LIN {X 0,Y 282.338,Z 551.265,A -85,B 0,C 180,E1 -17007.146,E2 -17007.146} C_VEL
LIN {X 0,Y 282.332,Z 551.855,A -85,B 0,C 180,E1 -17008.574,E2 -17008.574} C_VEL
LIN {X 0,Y 282.332,Z 551.855,A -85,B 0,C 180,E1 -17011.426,E2 -17011.426} C_VEL
LIN {X 0,Y 282.337,Z 551.265,A -85,B 0,C 180,E1 -17012.854,E2 -17012.854} C_VEL
LIN {X 0,Y 282.387,Z 548.814,A -85,B 0,C 180,E1 -17015.713,E2 -17015.713} C_VEL
LIN {X 0,Y 282.678,Z 545.862,A -85,B 0,C 180,E1 -17017.859,E2 -17017.859} C_VEL
LIN {X 0,Y 283.182,Z 541.872,A -85,B 0,C 180,E1 -17020.004,E2 -17020.004} C_VEL
LIN {X 0,Y 283.97,Z 536.74,A -85,B 0,C 180,E1 -17022.144,E2 -17022.144} C_VEL
LIN {X 0,Y 284.964,Z 531.479,A -85,B 0,C 180,E1 -17023.913,E2 -17023.913} C_VEL
LIN {X 0,Y 286.139,Z 525.162,A -85,B 0,C 180,E1 -17025.674,E2 -17025.674} C_VEL
LIN {X 0,Y 287.269,Z 519.212,A -85,B 0,C 180,E1 -17027.072,E2 -17027.072} C_VEL
LIN {X 0,Y 288.401,Z 512.283,A -85,B 0,C 180,E1 -17028.469,E2 -17028.469} C_VEL
LIN {X 0,Y 289.838,Z 504.105,A -85,B 0,C 180,E1 -17029.844,E2 -17029.844} C_VEL
LIN {X 0,Y 291.293,Z 495.598,A -85,B 0,C 180,E1 -17031.031,E2 -17031.031} C_VEL
LIN {X 0,Y 292.626,Z 486.885,A -85,B 0,C 180,E1 -17032.04,E2 -17032.04} C_VEL
LIN {X 0,Y 293.906,Z 477.128,A -85,B 0,C 180,E1 -17032.958,E2 -17032.958} C_VEL
LIN {X 0,Y 294.944,Z 468.339,A -85,B 0,C 180,E1 -17033.616,E2 -17033.616} C_VEL
LIN {X 0,Y 295.883,Z 458.415,A -85,B 0,C 180,E1 -17034.187,E2 -17034.187} C_VEL
LIN {X 0,Y 296.567,Z 448.566,A -85,B 0,C 180,E1 -17034.594,E2 -17034.594} C_VEL
LIN {X 0,Y 297.302,Z 424.442,A -85,B 0,C 180,E1 -17035.216,E2 -17035.216} C_VEL
LIN {X 0,Y 298.17,Z 386.954,A -85,B 0,C 180,E1 -17036.118,E2 -17036.118} C_VEL
LIN {X 0,Y 294.061,Z 364.054,A -85,B 0,C 180,E1 -17037.121,E2 -17037.121} C_VEL
LIN {X 0,Y 290.221,Z 346.945,A -85,B 0,C 180,E1 -17037.974,E2 -17037.974} C_VEL
LIN {X 0,Y 288.061,Z 341.163,A -85,B 0,C 180,E1 -17038.405,E2 -17038.405} C_VEL
LIN {X 0,Y 287.284,Z 336.939,A -85,B 0,C 180,E1 -17040.099,E2 -17040.099} C_VEL
LIN {X 0,Y 285.639,Z 328.615,A -85,B 0,C 180,E1 -17043.785,E2 -17043.785} C_VEL
LIN {X 0,Y 284.339,Z 322.594,A -85,B 0,C 180,E1 -17046.604,E2 -17046.604} C_VEL
LIN {X 0,Y 284.254,Z 322.548,A -85,B 0,C 180,E1 -17050.002,E2 -17050.002} C_VEL
LIN {X 0,Y 284.233,Z 322.579,A -85,B 0,C 180,E1 -17054.187,E2 -17054.187} C_VEL
LIN {X 0,Y 284.27,Z 322.574,A -85,B 0,C 180,E1 -17058.123,E2 -17058.123} C_VEL
LIN {X 0,Y 284.316,Z 322.57,A -85,B 0,C 180,E1 -17062.278,E2 -17062.278} C_VEL
LIN {X 0,Y 284.305,Z 322.55,A -85,B 0,C 180,E1 -17065.349,E2 -17065.349} C_VEL
LIN {X 0,Y 284.29,Z 322.571,A -85,B 0,C 180,E1 -17068.724,E2 -17068.724} C_VEL
LIN {X 0,Y 284.388,Z 322.531,A -85,B 0,C 180,E1 -17072.827,E2 -17072.827} C_VEL
LIN {X 0,Y 284.329,Z 322.564,A -85,B 0,C 180,E1 -17076.703,E2 -17076.703} C_VEL
LIN {X 0,Y 284.393,Z 322.523,A -85,B 0,C 180,E1 -17081.26,E2 -17081.26} C_VEL
LIN {X 0,Y 284.473,Z 322.542,A -85,B 0,C 180,E1 -17084.469,E2 -17084.469} C_VEL
LIN {X 0,Y 284.481,Z 322.525,A -85,B 0,C 180,E1 -17088.6,E2 -17088.6} C_VEL
LIN {X 0,Y 284.632,Z 322.493,A -85,B 0,C 180,E1 -17091.48,E2 -17091.48} C_VEL
LIN {X 0,Y 284.591,Z 322.532,A -85,B 0,C 180,E1 -17094.33,E2 -17094.33} C_VEL
LIN {X 0,Y 284.849,Z 322.475,A -85,B 0,C 180,E1 -17098.585,E2 -17098.585} C_VEL
LIN {X 0,Y 284.848,Z 322.466,A -85,B 0,C 180,E1 -17101.413,E2 -17101.413} C_VEL
LIN {X 0,Y 284.679,Z 322.513,A -85,B 0,C 180,E1 -17107.09,E2 -17107.09} C_VEL
LIN {X 0,Y 284.512,Z 322.504,A -85,B 0,C 180,E1 -17109.956,E2 -17109.956} C_VEL
LIN {X 0,Y 284.471,Z 322.549,A -85,B 0,C 180,E1 -17114.302,E2 -17114.302} C_VEL
LIN {X 0,Y 284.418,Z 322.539,A -85,B 0,C 180,E1 -17117.248,E2 -17117.248} C_VEL
LIN {X 0,Y 284.372,Z 322.535,A -85,B 0,C 180,E1 -17120.242,E2 -17120.242} C_VEL
LIN {X 0,Y 284.362,Z 322.562,A -85,B 0,C 180,E1 -17123.875,E2 -17123.875} C_VEL
LIN {X 0,Y 284.389,Z 322.532,A -85,B 0,C 180,E1 -17127.173,E2 -17127.173} C_VEL
LIN {X 0,Y 284.289,Z 322.574,A -85,B 0,C 180,E1 -17131.274,E2 -17131.274} C_VEL
LIN {X 0,Y 284.355,Z 322.546,A -85,B 0,C 180,E1 -17135.354,E2 -17135.354} C_VEL
LIN {X 0,Y 284.33,Z 322.57,A -85,B 0,C 180,E1 -17138.165,E2 -17138.165} C_VEL
LIN {X 0,Y 284.334,Z 322.56,A -85,B 0,C 180,E1 -17142.14,E2 -17142.14} C_VEL
LIN {X 0,Y 284.29,Z 322.533,A -85,B 0,C 180,E1 -17146.197,E2 -17146.197} C_VEL
LIN {X 0,Y 284.304,Z 322.538,A -85,B 0,C 180,E1 -17150.023,E2 -17150.023} C_VEL
LIN {X 0,Y 284.348,Z 322.545,A -85,B 0,C 180,E1 -17153.617,E2 -17153.617} C_VEL
LIN {X 0,Y 284.302,Z 322.553,A -85,B 0,C 180,E1 -17157.19,E2 -17157.19} C_VEL
LIN {X 0,Y 284.356,Z 322.708,A -85,B 0,C 180,E1 -17160.853,E2 -17160.853} C_VEL
LIN {X 0,Y 284.569,Z 323.646,A -85,B 0,C 180,E1 -17161.126,E2 -17161.126} C_VEL
LIN {X 0,Y 292.585,Z 338.677,A -85,B 0,C 180,E1 -17162.429,E2 -17162.429} C_VEL
LIN {X 0,Y 300.389,Z 349.784,A -85,B 0,C 180,E1 -17163.502,E2 -17163.502} C_VEL
LIN {X 0,Y 308.793,Z 359.275,A -85,B 0,C 180,E1 -17164.601,E2 -17164.601} C_VEL
LIN {X 0,Y 316.905,Z 367.975,A -85,B 0,C 180,E1 -17165.816,E2 -17165.816} C_VEL
LIN {X 0,Y 324.503,Z 375.523,A -85,B 0,C 180,E1 -17167.119,E2 -17167.119} C_VEL
LIN {X 0,Y 332.838,Z 383.472,A -85,B 0,C 180,E1 -17168.723,E2 -17168.723} C_VEL
LIN {X 0,Y 340.839,Z 390.558,A -85,B 0,C 180,E1 -17170.438,E2 -17170.438} C_VEL
LIN {X 0,Y 346.351,Z 394.989,A -85,B 0,C 180,E1 -17171.714,E2 -17171.714} C_VEL
LIN {X 0,Y 353.056,Z 400.728,A -85,B 0,C 180,E1 -17173.434,E2 -17173.434} C_VEL
LIN {X 0,Y 358.555,Z 404.823,A -85,B 0,C 180,E1 -17174.987,E2 -17174.987} C_VEL
LIN {X 0,Y 363.378,Z 408.762,A -85,B 0,C 180,E1 -17176.527,E2 -17176.527} C_VEL
LIN {X 0,Y 368.048,Z 411.828,A -85,B 0,C 180,E1 -17178.185,E2 -17178.185} C_VEL
LIN {X 0,Y 370.508,Z 413.424,A -85,B 0,C 180,E1 -17179.171,E2 -17179.171} C_VEL
LIN {X 0,Y 373.985,Z 416.445,A -85,B 0,C 180,E1 -17180.788,E2 -17180.788} C_VEL
LIN {X 0,Y 377.117,Z 418.611,A -85,B 0,C 180,E1 -17182.504,E2 -17182.504} C_VEL
LIN {X 0,Y 379.745,Z 420.059,A -85,B 0,C 180,E1 -17184.312,E2 -17184.312} C_VEL
LIN {X 0,Y 381.335,Z 420.74,A -85,B 0,C 180,E1 -17185.772,E2 -17185.772} C_VEL
LIN {X 0,Y 382.556,Z 421.148,A -85,B 0,C 180,E1 -17187.355,E2 -17187.355} C_VEL
LIN {X 0,Y 383.208,Z 421.566,A -85,B 0,C 180,E1 -17188.949,E2 -17188.949} C_VEL
LIN {X 0,Y 383.351,Z 421.508,A -85,B 0,C 180,E1 -17190,E2 -17190} C_VEL
LIN {X 0,Y 383.05,Z 421.431,A -85,B 0,C 180,E1 -17191.577,E2 -17191.577} C_VEL
LIN {X 0,Y 382.23,Z 420.939,A -85,B 0,C 180,E1 -17193.162,E2 -17193.162} C_VEL
LIN {X 0,Y 380.5,Z 420.427,A -85,B 0,C 180,E1 -17195.024,E2 -17195.024} C_VEL
LIN {X 0,Y 377.947,Z 419.106,A -85,B 0,C 180,E1 -17196.961,E2 -17196.961} C_VEL
LIN {X 0,Y 374.623,Z 416.948,A -85,B 0,C 180,E1 -17198.885,E2 -17198.885} C_VEL
LIN {X 0,Y 371.032,Z 413.897,A -85,B 0,C 180,E1 -17200.604,E2 -17200.604} C_VEL
LIN {X 0,Y 368.439,Z 411.979,A -85,B 0,C 180,E1 -17201.675,E2 -17201.675} C_VEL
LIN {X 0,Y 364.032,Z 409.248,A -85,B 0,C 180,E1 -17203.256,E2 -17203.256} C_VEL
LIN {X 0,Y 358.884,Z 405.11,A -85,B 0,C 180,E1 -17204.909,E2 -17204.909} C_VEL
LIN {X 0,Y 352.075,Z 399.957,A -85,B 0,C 180,E1 -17206.83,E2 -17206.83} C_VEL
LIN {X 0,Y 345.31,Z 394.26,A -85,B 0,C 180,E1 -17208.53,E2 -17208.53} C_VEL
LIN {X 0,Y 339.058,Z 388.935,A -85,B 0,C 180,E1 -17209.965,E2 -17209.965} C_VEL
LIN {X 0,Y 331.391,Z 382.051,A -85,B 0,C 180,E1 -17211.572,E2 -17211.572} C_VEL
LIN {X 0,Y 323.339,Z 374.346,A -85,B 0,C 180,E1 -17213.096,E2 -17213.096} C_VEL
LIN {X 0,Y 316.273,Z 367.284,A -85,B 0,C 180,E1 -17214.282,E2 -17214.282} C_VEL
LIN {X 0,Y 308.443,Z 358.947,A -85,B 0,C 180,E1 -17215.444,E2 -17215.444} C_VEL
LIN {X 0,Y 299.859,Z 349.077,A -85,B 0,C 180,E1 -17216.568,E2 -17216.568} C_VEL
LIN {X 0,Y 292.259,Z 338.141,A -85,B 0,C 180,E1 -17217.619,E2 -17217.619} C_VEL
LIN {X 0,Y 284.572,Z 323.628,A -85,B 0,C 180,E1 -17218.876,E2 -17218.876} C_VEL
LIN {X 0,Y 284.347,Z 322.628,A -85,B 0,C 180,E1 -17219.19,E2 -17219.19} C_VEL
LIN {X 0,Y 284.3,Z 322.55,A -85,B 0,C 180,E1 -17222.945,E2 -17222.945} C_VEL
LIN {X 0,Y 284.348,Z 322.545,A -85,B 0,C 180,E1 -17226.383,E2 -17226.383} C_VEL
LIN {X 0,Y 284.303,Z 322.537,A -85,B 0,C 180,E1 -17229.994,E2 -17229.994} C_VEL
LIN {X 0,Y 284.287,Z 322.541,A -85,B 0,C 180,E1 -17234.2,E2 -17234.2} C_VEL
LIN {X 0,Y 284.332,Z 322.558,A -85,B 0,C 180,E1 -17238.136,E2 -17238.136} C_VEL
LIN {X 0,Y 284.339,Z 322.567,A -85,B 0,C 180,E1 -17242.272,E2 -17242.272} C_VEL
LIN {X 0,Y 284.317,Z 322.548,A -85,B 0,C 180,E1 -17245.353,E2 -17245.353} C_VEL
LIN {X 0,Y 284.289,Z 322.574,A -85,B 0,C 180,E1 -17248.726,E2 -17248.726} C_VEL
LIN {X 0,Y 284.389,Z 322.532,A -85,B 0,C 180,E1 -17252.827,E2 -17252.827} C_VEL
LIN {X 0,Y 284.359,Z 322.565,A -85,B 0,C 180,E1 -17256.707,E2 -17256.707} C_VEL
LIN {X 0,Y 284.395,Z 322.526,A -85,B 0,C 180,E1 -17261.262,E2 -17261.262} C_VEL
LIN {X 0,Y 284.471,Z 322.547,A -85,B 0,C 180,E1 -17264.47,E2 -17264.47} C_VEL
LIN {X 0,Y 284.48,Z 322.518,A -85,B 0,C 180,E1 -17268.602,E2 -17268.602} C_VEL
LIN {X 0,Y 284.632,Z 322.5,A -85,B 0,C 180,E1 -17271.481,E2 -17271.481} C_VEL
LIN {X 0,Y 284.59,Z 322.533,A -85,B 0,C 180,E1 -17274.332,E2 -17274.332} C_VEL
LIN {X 0,Y 284.848,Z 322.467,A -85,B 0,C 180,E1 -17278.587,E2 -17278.587} C_VEL
LIN {X 0,Y 284.849,Z 322.475,A -85,B 0,C 180,E1 -17281.415,E2 -17281.415} C_VEL
LIN {X 0,Y 284.68,Z 322.508,A -85,B 0,C 180,E1 -17287.091,E2 -17287.091} C_VEL
LIN {X 0,Y 284.513,Z 322.504,A -85,B 0,C 180,E1 -17289.958,E2 -17289.958} C_VEL
LIN {X 0,Y 284.473,Z 322.548,A -85,B 0,C 180,E1 -17294.304,E2 -17294.304} C_VEL
LIN {X 0,Y 284.417,Z 322.529,A -85,B 0,C 180,E1 -17297.25,E2 -17297.25} C_VEL
LIN {X 0,Y 284.379,Z 322.536,A -85,B 0,C 180,E1 -17300.013,E2 -17300.013} C_VEL
LIN {X 0,Y 283.743,Z 322.631,A -85,B 0,C 180,E1 -17301.196,E2 -17301.196} C_VEL
LIN {X 0,Y 280.862,Z 322.997,A -85,B 0,C 180,E1 -17303.121,E2 -17303.121} C_VEL
LIN {X 0,Y 278.406,Z 323.292,A -85,B 0,C 180,E1 -17304.685,E2 -17304.685} C_VEL
LIN {X 0,Y 277.371,Z 323.408,A -85,B 0,C 180,E1 -17305.898,E2 -17305.898} C_VEL
LIN {X 0,Y 277.298,Z 323.414,A -85,B 0,C 180,E1 -17306.309,E2 -17306.309} C_VEL
LIN {X 0,Y 277.269,Z 323.449,A -85,B 0,C 180,E1 -17310.483,E2 -17310.483} C_VEL
LIN {X 0,Y 277.244,Z 323.427,A -85,B 0,C 180,E1 -17313.897,E2 -17313.897} C_VEL
LIN {X 0,Y 277.262,Z 323.448,A -85,B 0,C 180,E1 -17317.471,E2 -17317.471} C_VEL
LIN {X 0,Y 277.208,Z 323.449,A -85,B 0,C 180,E1 -17321.238,E2 -17321.238} C_VEL
LIN {X 0,Y 277.194,Z 323.451,A -85,B 0,C 180,E1 -17325.229,E2 -17325.229} C_VEL
LIN {X 0,Y 277.176,Z 323.43,A -85,B 0,C 180,E1 -17328.759,E2 -17328.759} C_VEL
LIN {X 0,Y 277.301,Z 323.586,A -85,B 0,C 180,E1 -17332.902,E2 -17332.902} C_VEL
LIN {X 0,Y 278.886,Z 330.791,A -85,B 0,C 180,E1 -17336.331,E2 -17336.331} C_VEL
LIN {X 0,Y 280.435,Z 338.656,A -85,B 0,C 180,E1 -17339.92,E2 -17339.92} C_VEL
LIN {X 0,Y 280.841,Z 340.955,A -85,B 0,C 180,E1 -17340.795,E2 -17340.795} C_VEL
LIN {X 0,Y 284.504,Z 350.337,A -85,B 0,C 180,E1 -17341.513,E2 -17341.513} C_VEL
LIN {X 0,Y 289.328,Z 373.325,A -85,B 0,C 180,E1 -17342.656,E2 -17342.656} C_VEL
LIN {X 0,Y 291.893,Z 388.914,A -85,B 0,C 180,E1 -17343.334,E2 -17343.334} C_VEL
LIN {X 0,Y 290.229,Z 447.041,A -85,B 0,C 180,E1 -17344.784,E2 -17344.784} C_VEL
LIN {X 0,Y 289.511,Z 457.348,A -85,B 0,C 180,E1 -17345.197,E2 -17345.197} C_VEL
LIN {X 0,Y 288.58,Z 466.857,A -85,B 0,C 180,E1 -17345.735,E2 -17345.735} C_VEL
LIN {X 0,Y 287.504,Z 475.928,A -85,B 0,C 180,E1 -17346.405,E2 -17346.405} C_VEL
LIN {X 0,Y 286.312,Z 485.06,A -85,B 0,C 180,E1 -17347.257,E2 -17347.257} C_VEL
LIN {X 0,Y 284.893,Z 494.052,A -85,B 0,C 180,E1 -17348.283,E2 -17348.283} C_VEL
LIN {X 0,Y 283.36,Z 502.776,A -85,B 0,C 180,E1 -17349.493,E2 -17349.493} C_VEL
LIN {X 0,Y 281.983,Z 510.168,A -85,B 0,C 180,E1 -17350.717,E2 -17350.717} C_VEL
LIN {X 0,Y 280.589,Z 518.247,A -85,B 0,C 180,E1 -17352.331,E2 -17352.331} C_VEL
LIN {X 0,Y 279.246,Z 524.966,A -85,B 0,C 180,E1 -17353.928,E2 -17353.928} C_VEL
LIN {X 0,Y 278.035,Z 531.284,A -85,B 0,C 180,E1 -17355.733,E2 -17355.733} C_VEL
LIN {X 0,Y 276.992,Z 536.544,A -85,B 0,C 180,E1 -17357.546,E2 -17357.546} C_VEL
LIN {X 0,Y 276.172,Z 541.677,A -85,B 0,C 180,E1 -17359.739,E2 -17359.739} C_VEL
LIN {X 0,Y 275.608,Z 545.667,A -85,B 0,C 180,E1 -17361.938,E2 -17361.938} C_VEL
LIN {X 0,Y 275.254,Z 549.304,A -85,B 0,C 180,E1 -17364.741,E2 -17364.741} C_VEL
LIN {X 0,Y 275.247,Z 551.071,A -85,B 0,C 180,E1 -17367.073,E2 -17367.073} C_VEL
LIN {X 0,Y 275.256,Z 551.662,A -85,B 0,C 180,E1 -17368.537,E2 -17368.537} C_VEL
LIN {X 0,Y 275.256,Z 551.662,A -85,B 0,C 180,E1 -17371.463,E2 -17371.463} C_VEL
LIN {X 0,Y 275.246,Z 551.071,A -85,B 0,C 180,E1 -17372.927,E2 -17372.927} C_VEL
LIN {X 0,Y 275.3,Z 548.619,A -85,B 0,C 180,E1 -17375.861,E2 -17375.861} C_VEL
LIN {X 0,Y 275.607,Z 545.667,A -85,B 0,C 180,E1 -17378.062,E2 -17378.062} C_VEL
LIN {X 0,Y 276.172,Z 541.677,A -85,B 0,C 180,E1 -17380.261,E2 -17380.261} C_VEL
LIN {X 0,Y 276.992,Z 536.544,A -85,B 0,C 180,E1 -17382.454,E2 -17382.454} C_VEL
LIN {X 0,Y 278.03,Z 531.284,A -85,B 0,C 180,E1 -17384.268,E2 -17384.268} C_VEL
LIN {X 0,Y 279.263,Z 524.967,A -85,B 0,C 180,E1 -17386.071,E2 -17386.071} C_VEL
LIN {X 0,Y 280.665,Z 518.016,A -85,B 0,C 180,E1 -17387.718,E2 -17387.718} C_VEL
LIN {X 0,Y 281.664,Z 512.088,A -85,B 0,C 180,E1 -17388.927,E2 -17388.927} C_VEL
LIN {X 0,Y 283.167,Z 503.911,A -85,B 0,C 180,E1 -17390.332,E2 -17390.332} C_VEL
LIN {X 0,Y 284.677,Z 495.404,A -85,B 0,C 180,E1 -17391.544,E2 -17391.544} C_VEL
LIN {X 0,Y 286.062,Z 486.691,A -85,B 0,C 180,E1 -17392.573,E2 -17392.573} C_VEL
LIN {X 0,Y 287.374,Z 476.934,A -85,B 0,C 180,E1 -17393.511,E2 -17393.511} C_VEL
LIN {X 0,Y 288.451,Z 468.145,A -85,B 0,C 180,E1 -17394.181,E2 -17394.181} C_VEL
LIN {X 0,Y 289.426,Z 458.221,A -85,B 0,C 180,E1 -17394.763,E2 -17394.763} C_VEL
LIN {X 0,Y 290.134,Z 448.372,A -85,B 0,C 180,E1 -17395.177,E2 -17395.177} C_VEL
LIN {X 0,Y 290.91,Z 424.264,A -85,B 0,C 180,E1 -17395.81,E2 -17395.81} C_VEL
LIN {X 0,Y 291.819,Z 388.268,A -85,B 0,C 180,E1 -17396.69,E2 -17396.69} C_VEL
LIN {X 0,Y 288.062,Z 366.799,A -85,B 0,C 180,E1 -17397.653,E2 -17397.653} C_VEL
LIN {X 0,Y 284.215,Z 349.549,A -85,B 0,C 180,E1 -17398.54,E2 -17398.54} C_VEL
LIN {X 0,Y 280.84,Z 340.923,A -85,B 0,C 180,E1 -17399.208,E2 -17399.208} C_VEL
LIN {X 0,Y 279.86,Z 335.827,A -85,B 0,C 180,E1 -17401.368,E2 -17401.368} C_VEL
LIN {X 0,Y 278.214,Z 327.795,A -85,B 0,C 180,E1 -17405.077,E2 -17405.077} C_VEL
LIN {X 0,Y 277.285,Z 323.452,A -85,B 0,C 180,E1 -17407.256,E2 -17407.256} C_VEL
LIN {X 0,Y 277.176,Z 323.43,A -85,B 0,C 180,E1 -17411.241,E2 -17411.241} C_VEL
LIN {X 0,Y 277.197,Z 323.447,A -85,B 0,C 180,E1 -17415.226,E2 -17415.226} C_VEL
LIN {X 0,Y 277.22,Z 323.44,A -85,B 0,C 180,E1 -17419.511,E2 -17419.511} C_VEL
LIN {X 0,Y 277.262,Z 323.448,A -85,B 0,C 180,E1 -17422.529,E2 -17422.529} C_VEL
LIN {X 0,Y 277.244,Z 323.427,A -85,B 0,C 180,E1 -17426.103,E2 -17426.103} C_VEL
LIN {X 0,Y 277.259,Z 323.451,A -85,B 0,C 180,E1 -17429.537,E2 -17429.537} C_VEL
LIN {X 0,Y 277.35,Z 323.407,A -85,B 0,C 180,E1 -17432.862,E2 -17432.862} C_VEL
LIN {X 0,Y 277.292,Z 323.44,A -85,B 0,C 180,E1 -17436.075,E2 -17436.075} C_VEL
LIN {X 0,Y 277.337,Z 323.404,A -85,B 0,C 180,E1 -17440.765,E2 -17440.765} C_VEL
LIN {X 0,Y 277.423,Z 323.424,A -85,B 0,C 180,E1 -17445.324,E2 -17445.324} C_VEL
LIN {X 0,Y 277.455,Z 323.383,A -85,B 0,C 180,E1 -17449.786,E2 -17449.786} C_VEL
LIN {X 0,Y 277.634,Z 323.384,A -85,B 0,C 180,E1 -17452.728,E2 -17452.728} C_VEL
LIN {X 0,Y 277.815,Z 323.351,A -85,B 0,C 180,E1 -17458.55,E2 -17458.55} C_VEL
LIN {X 0,Y 277.814,Z 323.342,A -85,B 0,C 180,E1 -17461.449,E2 -17461.449} C_VEL
LIN {X 0,Y 277.634,Z 323.389,A -85,B 0,C 180,E1 -17467.271,E2 -17467.271} C_VEL
LIN {X 0,Y 277.454,Z 323.382,A -85,B 0,C 180,E1 -17470.212,E2 -17470.212} C_VEL
LIN {X 0,Y 277.421,Z 323.429,A -85,B 0,C 180,E1 -17474.674,E2 -17474.674} C_VEL
LIN {X 0,Y 277.337,Z 323.404,A -85,B 0,C 180,E1 -17479.233,E2 -17479.233} C_VEL
LIN {X 0,Y 277.312,Z 323.441,A -85,B 0,C 180,E1 -17484.17,E2 -17484.17} C_VEL
LIN {X 0,Y 277.318,Z 323.412,A -85,B 0,C 180,E1 -17487.504,E2 -17487.504} C_VEL
LIN {X 0,Y 277.265,Z 323.446,A -85,B 0,C 180,E1 -17490.481,E2 -17490.481} C_VEL
LIN {X 0,Y 277.247,Z 323.43,A -85,B 0,C 180,E1 -17493.895,E2 -17493.895} C_VEL
LIN {X 0,Y 277.284,Z 323.447,A -85,B 0,C 180,E1 -17497.466,E2 -17497.466} C_VEL
LIN {X 0,Y 277.257,Z 323.432,A -85,B 0,C 180,E1 -17501.227,E2 -17501.227} C_VEL
LIN {X 0,Y 277.236,Z 323.431,A -85,B 0,C 180,E1 -17505.218,E2 -17505.218} C_VEL
LIN {X 0,Y 277.221,Z 323.408,A -85,B 0,C 180,E1 -17509.511,E2 -17509.511} C_VEL
LIN {X 0,Y 277.281,Z 323.445,A -85,B 0,C 180,E1 -17512.534,E2 -17512.534} C_VEL
LIN {X 0,Y 277.249,Z 323.415,A -85,B 0,C 180,E1 -17516.105,E2 -17516.105} C_VEL
LIN {X 0,Y 277.305,Z 323.576,A -85,B 0,C 180,E1 -17520.073,E2 -17520.073} C_VEL
LIN {X 0,Y 277.556,Z 324.569,A -85,B 0,C 180,E1 -17520.348,E2 -17520.348} C_VEL
LIN {X 0,Y 287.343,Z 342.912,A -85,B 0,C 180,E1 -17521.996,E2 -17521.996} C_VEL
LIN {X 0,Y 294.758,Z 353.585,A -85,B 0,C 180,E1 -17523.052,E2 -17523.052} C_VEL
LIN {X 0,Y 304.118,Z 364.334,A -85,B 0,C 180,E1 -17524.244,E2 -17524.244} C_VEL
LIN {X 0,Y 311.901,Z 372.421,A -85,B 0,C 180,E1 -17525.315,E2 -17525.315} C_VEL
LIN {X 0,Y 318.089,Z 378.443,A -85,B 0,C 180,E1 -17526.266,E2 -17526.266} C_VEL
LIN {X 0,Y 324.451,Z 384.567,A -85,B 0,C 180,E1 -17527.372,E2 -17527.372} C_VEL
LIN {X 0,Y 332.426,Z 391.897,A -85,B 0,C 180,E1 -17528.906,E2 -17528.906} C_VEL
LIN {X 0,Y 340.748,Z 399.068,A -85,B 0,C 180,E1 -17530.692,E2 -17530.692} C_VEL
LIN {X 0,Y 346.278,Z 403.439,A -85,B 0,C 180,E1 -17531.979,E2 -17531.979} C_VEL
LIN {X 0,Y 352.189,Z 408.23,A -85,B 0,C 180,E1 -17533.492,E2 -17533.492} C_VEL
LIN {X 0,Y 356.757,Z 411.554,A -85,B 0,C 180,E1 -17534.763,E2 -17534.763} C_VEL
LIN {X 0,Y 361.884,Z 415.618,A -85,B 0,C 180,E1 -17536.362,E2 -17536.362} C_VEL
LIN {X 0,Y 366.483,Z 418.608,A -85,B 0,C 180,E1 -17537.961,E2 -17537.961} C_VEL
LIN {X 0,Y 369.009,Z 420.209,A -85,B 0,C 180,E1 -17538.942,E2 -17538.942} C_VEL
LIN {X 0,Y 372.659,Z 423.307,A -85,B 0,C 180,E1 -17540.597,E2 -17540.597} C_VEL
LIN {X 0,Y 375.863,Z 425.477,A -85,B 0,C 180,E1 -17542.306,E2 -17542.306} C_VEL
LIN {X 0,Y 378.844,Z 427.104,A -85,B 0,C 180,E1 -17544.299,E2 -17544.299} C_VEL
LIN {X 0,Y 380.515,Z 427.791,A -85,B 0,C 180,E1 -17545.829,E2 -17545.829} C_VEL
LIN {X 0,Y 381.686,Z 428.196,A -85,B 0,C 180,E1 -17547.349,E2 -17547.349} C_VEL
LIN {X 0,Y 382.346,Z 428.597,A -85,B 0,C 180,E1 -17548.947,E2 -17548.947} C_VEL
LIN {X 0,Y 382.488,Z 428.54,A -85,B 0,C 180,E1 -17550,E2 -17550} C_VEL
LIN {X 0,Y 382.181,Z 428.48,A -85,B 0,C 180,E1 -17551.581,E2 -17551.581} C_VEL
LIN {X 0,Y 381.093,Z 427.919,A -85,B 0,C 180,E1 -17553.514,E2 -17553.514} C_VEL
LIN {X 0,Y 379.012,Z 427.165,A -85,B 0,C 180,E1 -17555.563,E2 -17555.563} C_VEL
LIN {X 0,Y 376.179,Z 425.679,A -85,B 0,C 180,E1 -17557.514,E2 -17557.514} C_VEL
LIN {X 0,Y 372.829,Z 423.468,A -85,B 0,C 180,E1 -17559.32,E2 -17559.32} C_VEL
LIN {X 0,Y 369.009,Z 420.204,A -85,B 0,C 180,E1 -17561.058,E2 -17561.058} C_VEL
LIN {X 0,Y 363.501,Z 416.773,A -85,B 0,C 180,E1 -17563.102,E2 -17563.102} C_VEL
LIN {X 0,Y 357.89,Z 412.57,A -85,B 0,C 180,E1 -17564.891,E2 -17564.891} C_VEL
LIN {X 0,Y 353.91,Z 409.438,A -85,B 0,C 180,E1 -17566.037,E2 -17566.037} C_VEL
LIN {X 0,Y 348.023,Z 404.978,A -85,B 0,C 180,E1 -17567.589,E2 -17567.589} C_VEL
LIN {X 0,Y 342.613,Z 400.499,A -85,B 0,C 180,E1 -17568.892,E2 -17568.892} C_VEL
LIN {X 0,Y 336.047,Z 394.971,A -85,B 0,C 180,E1 -17570.342,E2 -17570.342} C_VEL
LIN {X 0,Y 328.448,Z 388.318,A -85,B 0,C 180,E1 -17571.882,E2 -17571.882} C_VEL
LIN {X 0,Y 319.943,Z 380.342,A -85,B 0,C 180,E1 -17573.421,E2 -17573.421} C_VEL
LIN {X 0,Y 312.089,Z 372.639,A -85,B 0,C 180,E1 -17574.656,E2 -17574.656} C_VEL
LIN {X 0,Y 303.673,Z 363.897,A -85,B 0,C 180,E1 -17575.811,E2 -17575.811} C_VEL
LIN {X 0,Y 294.558,Z 353.322,A -85,B 0,C 180,E1 -17576.975,E2 -17576.975} C_VEL
LIN {X 0,Y 287.007,Z 342.377,A -85,B 0,C 180,E1 -17578.055,E2 -17578.055} C_VEL
LIN {X 0,Y 277.549,Z 324.574,A -85,B 0,C 180,E1 -17579.65,E2 -17579.65} C_VEL
LIN {X 0,Y 277.3,Z 323.521,A -85,B 0,C 180,E1 -17579.964,E2 -17579.964} C_VEL
LIN {X 0,Y 277.249,Z 323.415,A -85,B 0,C 180,E1 -17583.895,E2 -17583.895} C_VEL
LIN {X 0,Y 277.281,Z 323.445,A -85,B 0,C 180,E1 -17587.466,E2 -17587.466} C_VEL
LIN {X 0,Y 277.211,Z 323.4,A -85,B 0,C 180,E1 -17591.235,E2 -17591.235} C_VEL
LIN {X 0,Y 277.24,Z 323.44,A -85,B 0,C 180,E1 -17595.217,E2 -17595.217} C_VEL
LIN {X 0,Y 277.288,Z 323.427,A -85,B 0,C 180,E1 -17599.495,E2 -17599.495} C_VEL
LIN {X 0,Y 277.284,Z 323.447,A -85,B 0,C 180,E1 -17602.534,E2 -17602.534} C_VEL
LIN {X 0,Y 277.247,Z 323.43,A -85,B 0,C 180,E1 -17606.105,E2 -17606.105} C_VEL
LIN {X 0,Y 277.255,Z 323.448,A -85,B 0,C 180,E1 -17609.539,E2 -17609.539} C_VEL
LIN {X 0,Y 277.351,Z 323.408,A -85,B 0,C 180,E1 -17612.864,E2 -17612.864} C_VEL
LIN {X 0,Y 277.322,Z 323.439,A -85,B 0,C 180,E1 -17616.08,E2 -17616.08} C_VEL
LIN {X 0,Y 277.337,Z 323.404,A -85,B 0,C 180,E1 -17620.767,E2 -17620.767} C_VEL
LIN {X 0,Y 277.421,Z 323.429,A -85,B 0,C 180,E1 -17625.326,E2 -17625.326} C_VEL
LIN {X 0,Y 277.454,Z 323.382,A -85,B 0,C 180,E1 -17629.788,E2 -17629.788} C_VEL
LIN {X 0,Y 277.634,Z 323.389,A -85,B 0,C 180,E1 -17632.729,E2 -17632.729} C_VEL
LIN {X 0,Y 277.814,Z 323.342,A -85,B 0,C 180,E1 -17638.551,E2 -17638.551} C_VEL
LIN {X 0,Y 277.815,Z 323.351,A -85,B 0,C 180,E1 -17641.45,E2 -17641.45} C_VEL
LIN {X 0,Y 277.634,Z 323.384,A -85,B 0,C 180,E1 -17647.272,E2 -17647.272} C_VEL
LIN {X 0,Y 277.455,Z 323.383,A -85,B 0,C 180,E1 -17650.214,E2 -17650.214} C_VEL
LIN {X 0,Y 277.423,Z 323.424,A -85,B 0,C 180,E1 -17654.676,E2 -17654.676} C_VEL
LIN {X 0,Y 277.337,Z 323.404,A -85,B 0,C 180,E1 -17659.235,E2 -17659.235} C_VEL
LIN {X 0,Y 277.287,Z 323.437,A -85,B 0,C 180,E1 -17664.158,E2 -17664.158} C_VEL
LIN {X 0,Y 277.298,Z 323.414,A -85,B 0,C 180,E1 -17666.309,E2 -17666.309} C_VEL
LIN {X 0,Y 276.64,Z 323.5,A -85,B 0,C 180,E1 -17667.521,E2 -17667.521} C_VEL
LIN {X 0,Y 273.725,Z 323.885,A -85,B 0,C 180,E1 -17669.493,E2 -17669.493} C_VEL
LIN {X 0,Y 271.261,Z 324.194,A -85,B 0,C 180,E1 -17671.096,E2 -17671.096} C_VEL
LIN {X 0,Y 270.239,Z 324.311,A -85,B 0,C 180,E1 -17672.34,E2 -17672.34} C_VEL
LIN {X 0,Y 270.176,Z 324.312,A -85,B 0,C 180,E1 -17672.762,E2 -17672.762} C_VEL
LIN {X 0,Y 270.213,Z 324.327,A -85,B 0,C 180,E1 -17676.743,E2 -17676.743} C_VEL
LIN {X 0,Y 270.167,Z 324.322,A -85,B 0,C 180,E1 -17681.029,E2 -17681.029} C_VEL
LIN {X 0,Y 270.149,Z 324.324,A -85,B 0,C 180,E1 -17684.622,E2 -17684.622} C_VEL
LIN {X 0,Y 270.15,Z 324.322,A -85,B 0,C 180,E1 -17687.439,E2 -17687.439} C_VEL
LIN {X 0,Y 270.232,Z 324.445,A -85,B 0,C 180,E1 -17692.268,E2 -17692.268} C_VEL
LIN {X 0,Y 271.818,Z 331.673,A -85,B 0,C 180,E1 -17695.831,E2 -17695.831} C_VEL
LIN {X 0,Y 273.551,Z 340.382,A -85,B 0,C 180,E1 -17699.864,E2 -17699.864} C_VEL
LIN {X 0,Y 274.114,Z 342.282,A -85,B 0,C 180,E1 -17700.096,E2 -17700.096} C_VEL
LIN {X 0,Y 278.471,Z 352.731,A -85,B 0,C 180,E1 -17700.912,E2 -17700.912} C_VEL
LIN {X 0,Y 282.694,Z 372.939,A -85,B 0,C 180,E1 -17701.953,E2 -17701.953} C_VEL
LIN {X 0,Y 285.509,Z 390.044,A -85,B 0,C 180,E1 -17702.726,E2 -17702.726} C_VEL
LIN {X 0,Y 283.834,Z 446.854,A -85,B 0,C 180,E1 -17704.175,E2 -17704.175} C_VEL
LIN {X 0,Y 283.089,Z 457.154,A -85,B 0,C 180,E1 -17704.595,E2 -17704.595} C_VEL
LIN {X 0,Y 282.111,Z 466.663,A -85,B 0,C 180,E1 -17705.141,E2 -17705.141} C_VEL
LIN {X 0,Y 281.016,Z 475.734,A -85,B 0,C 180,E1 -17705.826,E2 -17705.826} C_VEL
LIN {X 0,Y 279.764,Z 484.865,A -85,B 0,C 180,E1 -17706.694,E2 -17706.694} C_VEL
LIN {X 0,Y 278.292,Z 493.858,A -85,B 0,C 180,E1 -17707.741,E2 -17707.741} C_VEL
LIN {X 0,Y 276.716,Z 502.582,A -85,B 0,C 180,E1 -17708.977,E2 -17708.977} C_VEL
LIN {X 0,Y 275.282,Z 509.974,A -85,B 0,C 180,E1 -17710.229,E2 -17710.229} C_VEL
LIN {X 0,Y 273.816,Z 517.499,A -85,B 0,C 180,E1 -17711.748,E2 -17711.748} C_VEL
LIN {X 0,Y 272.723,Z 523.397,A -85,B 0,C 180,E1 -17713.148,E2 -17713.148} C_VEL
LIN {X 0,Y 271.41,Z 529.934,A -85,B 0,C 180,E1 -17714.993,E2 -17714.993} C_VEL
LIN {X 0,Y 270.425,Z 534.434,A -85,B 0,C 180,E1 -17716.474,E2 -17716.474} C_VEL
LIN {X 0,Y 269.417,Z 539.928,A -85,B 0,C 180,E1 -17718.718,E2 -17718.718} C_VEL
LIN {X 0,Y 268.727,Z 544.255,A -85,B 0,C 180,E1 -17720.972,E2 -17720.972} C_VEL
LIN {X 0,Y 268.419,Z 546.624,A -85,B 0,C 180,E1 -17722.478,E2 -17722.478} C_VEL
LIN {X 0,Y 268.167,Z 549.278,A -85,B 0,C 180,E1 -17724.809,E2 -17724.809} C_VEL
LIN {X 0,Y 268.159,Z 550.878,A -85,B 0,C 180,E1 -17726.995,E2 -17726.995} C_VEL
LIN {X 0,Y 268.182,Z 551.469,A -85,B 0,C 180,E1 -17728.498,E2 -17728.498} C_VEL
LIN {X 0,Y 268.182,Z 551.469,A -85,B 0,C 180,E1 -17731.502,E2 -17731.502} C_VEL
LIN {X 0,Y 268.157,Z 550.878,A -85,B 0,C 180,E1 -17733.005,E2 -17733.005} C_VEL
LIN {X 0,Y 268.225,Z 548.425,A -85,B 0,C 180,E1 -17736.016,E2 -17736.016} C_VEL
LIN {X 0,Y 268.554,Z 545.473,A -85,B 0,C 180,E1 -17738.275,E2 -17738.275} C_VEL
LIN {X 0,Y 269.158,Z 541.482,A -85,B 0,C 180,E1 -17740.531,E2 -17740.531} C_VEL
LIN {X 0,Y 270.032,Z 536.35,A -85,B 0,C 180,E1 -17742.781,E2 -17742.781} C_VEL
LIN {X 0,Y 271.127,Z 531.089,A -85,B 0,C 180,E1 -17744.639,E2 -17744.639} C_VEL
LIN {X 0,Y 272.415,Z 524.772,A -85,B 0,C 180,E1 -17746.486,E2 -17746.486} C_VEL
LIN {X 0,Y 273.662,Z 518.823,A -85,B 0,C 180,E1 -17747.949,E2 -17747.949} C_VEL
LIN {X 0,Y 274.933,Z 511.894,A -85,B 0,C 180,E1 -17749.409,E2 -17749.409} C_VEL
LIN {X 0,Y 276.491,Z 503.716,A -85,B 0,C 180,E1 -17750.846,E2 -17750.846} C_VEL
LIN {X 0,Y 278.066,Z 495.209,A -85,B 0,C 180,E1 -17752.083,E2 -17752.083} C_VEL
LIN {X 0,Y 279.517,Z 486.497,A -85,B 0,C 180,E1 -17753.132,E2 -17753.132} C_VEL
LIN {X 0,Y 280.875,Z 476.74,A -85,B 0,C 180,E1 -17754.089,E2 -17754.089} C_VEL
LIN {X 0,Y 281.989,Z 467.951,A -85,B 0,C 180,E1 -17754.772,E2 -17754.772} C_VEL
LIN {X 0,Y 283.005,Z 458.028,A -85,B 0,C 180,E1 -17755.364,E2 -17755.364} C_VEL
LIN {X 0,Y 283.741,Z 448.179,A -85,B 0,C 180,E1 -17755.785,E2 -17755.785} C_VEL
LIN {X 0,Y 284.54,Z 424.228,A -85,B 0,C 180,E1 -17756.428,E2 -17756.428} C_VEL
LIN {X 0,Y 285.411,Z 388.541,A -85,B 0,C 180,E1 -17757.326,E2 -17757.326} C_VEL
LIN {X 0,Y 281.506,Z 366.746,A -85,B 0,C 180,E1 -17758.35,E2 -17758.35} C_VEL
LIN {X 0,Y 278.144,Z 351.763,A -85,B 0,C 180,E1 -17759.153,E2 -17759.153} C_VEL
LIN {X 0,Y 273.667,Z 340.943,A -85,B 0,C 180,E1 -17760.022,E2 -17760.022} C_VEL
LIN {X 0,Y 273.458,Z 340.123,A -85,B 0,C 180,E1 -17760.225,E2 -17760.225} C_VEL
LIN {X 0,Y 271.819,Z 331.672,A -85,B 0,C 180,E1 -17764.169,E2 -17764.169} C_VEL
LIN {X 0,Y 270.226,Z 324.402,A -85,B 0,C 180,E1 -17767.792,E2 -17767.792} C_VEL
LIN {X 0,Y 270.15,Z 324.323,A -85,B 0,C 180,E1 -17772.561,E2 -17772.561} C_VEL
LIN {X 0,Y 270.164,Z 324.329,A -85,B 0,C 180,E1 -17776.75,E2 -17776.75} C_VEL
LIN {X 0,Y 270.196,Z 324.319,A -85,B 0,C 180,E1 -17781.288,E2 -17781.288} C_VEL
LIN {X 0,Y 270.199,Z 324.308,A -85,B 0,C 180,E1 -17785.093,E2 -17785.093} C_VEL
LIN {X 0,Y 270.198,Z 324.328,A -85,B 0,C 180,E1 -17789.129,E2 -17789.129} C_VEL
LIN {X 0,Y 270.259,Z 324.295,A -85,B 0,C 180,E1 -17792.145,E2 -17792.145} C_VEL
LIN {X 0,Y 270.233,Z 324.312,A -85,B 0,C 180,E1 -17795.537,E2 -17795.537} C_VEL
LIN {X 0,Y 270.295,Z 324.285,A -85,B 0,C 180,E1 -17800.243,E2 -17800.243} C_VEL
LIN {X 0,Y 270.391,Z 324.297,A -85,B 0,C 180,E1 -17804.934,E2 -17804.934} C_VEL
LIN {X 0,Y 270.407,Z 324.263,A -85,B 0,C 180,E1 -17809.517,E2 -17809.517} C_VEL
LIN {X 0,Y 270.593,Z 324.256,A -85,B 0,C 180,E1 -17812.538,E2 -17812.538} C_VEL
LIN {X 0,Y 270.781,Z 324.227,A -85,B 0,C 180,E1 -17818.512,E2 -17818.512} C_VEL
LIN {X 0,Y 270.78,Z 324.218,A -85,B 0,C 180,E1 -17821.486,E2 -17821.486} C_VEL
LIN {X 0,Y 270.592,Z 324.264,A -85,B 0,C 180,E1 -17827.461,E2 -17827.461} C_VEL
LIN {X 0,Y 270.406,Z 324.26,A -85,B 0,C 180,E1 -17830.482,E2 -17830.482} C_VEL
LIN {X 0,Y 270.39,Z 324.305,A -85,B 0,C 180,E1 -17835.064,E2 -17835.064} C_VEL
LIN {X 0,Y 270.295,Z 324.282,A -85,B 0,C 180,E1 -17839.755,E2 -17839.755} C_VEL
LIN {X 0,Y 270.267,Z 324.315,A -85,B 0,C 180,E1 -17844.585,E2 -17844.585} C_VEL
LIN {X 0,Y 270.264,Z 324.291,A -85,B 0,C 180,E1 -17847.908,E2 -17847.908} C_VEL
LIN {X 0,Y 270.178,Z 324.331,A -85,B 0,C 180,E1 -17851.348,E2 -17851.348} C_VEL
LIN {X 0,Y 270.209,Z 324.304,A -85,B 0,C 180,E1 -17854.903,E2 -17854.903} C_VEL
LIN {X 0,Y 270.216,Z 324.322,A -85,B 0,C 180,E1 -17858.717,E2 -17858.717} C_VEL
LIN {X 0,Y 270.216,Z 324.322,A -85,B 0,C 180,E1 -17862.548,E2 -17862.548} C_VEL
LIN {X 0,Y 270.183,Z 324.279,A -85,B 0,C 180,E1 -17866.746,E2 -17866.746} C_VEL
LIN {X 0,Y 270.204,Z 324.324,A -85,B 0,C 180,E1 -17871.375,E2 -17871.375} C_VEL
LIN {X 0,Y 270.21,Z 324.289,A -85,B 0,C 180,E1 -17875.097,E2 -17875.097} C_VEL
LIN {X 0,Y 270.246,Z 324.545,A -85,B 0,C 180,E1 -17879.292,E2 -17879.292} C_VEL
LIN {X 0,Y 270.528,Z 325.667,A -85,B 0,C 180,E1 -17879.535,E2 -17879.535} C_VEL
LIN {X 0,Y 282.699,Z 348.129,A -85,B 0,C 180,E1 -17881.638,E2 -17881.638} C_VEL
LIN {X 0,Y 290.789,Z 359.59,A -85,B 0,C 180,E1 -17882.814,E2 -17882.814} C_VEL
LIN {X 0,Y 300.397,Z 370.35,A -85,B 0,C 180,E1 -17884.04,E2 -17884.04} C_VEL
LIN {X 0,Y 308.857,Z 379.072,A -85,B 0,C 180,E1 -17885.14,E2 -17885.14} C_VEL
LIN {X 0,Y 317.797,Z 387.589,A -85,B 0,C 180,E1 -17886.488,E2 -17886.488} C_VEL
LIN {X 0,Y 326.083,Z 395.114,A -85,B 0,C 180,E1 -17887.935,E2 -17887.935} C_VEL
LIN {X 0,Y 334.469,Z 402.342,A -85,B 0,C 180,E1 -17889.596,E2 -17889.596} C_VEL
LIN {X 0,Y 341.112,Z 407.621,A -85,B 0,C 180,E1 -17891.037,E2 -17891.037} C_VEL
LIN {X 0,Y 348.41,Z 413.557,A -85,B 0,C 180,E1 -17892.801,E2 -17892.801} C_VEL
LIN {X 0,Y 355.223,Z 418.552,A -85,B 0,C 180,E1 -17894.623,E2 -17894.623} C_VEL
LIN {X 0,Y 360.743,Z 422.782,A -85,B 0,C 180,E1 -17896.318,E2 -17896.318} C_VEL
LIN {X 0,Y 365.559,Z 425.735,A -85,B 0,C 180,E1 -17897.974,E2 -17897.974} C_VEL
LIN {X 0,Y 367.771,Z 427.262,A -85,B 0,C 180,E1 -17898.832,E2 -17898.832} C_VEL
LIN {X 0,Y 371.676,Z 430.424,A -85,B 0,C 180,E1 -17900.572,E2 -17900.572} C_VEL
LIN {X 0,Y 374.925,Z 432.543,A -85,B 0,C 180,E1 -17902.286,E2 -17902.286} C_VEL
LIN {X 0,Y 377.939,Z 434.149,A -85,B 0,C 180,E1 -17904.285,E2 -17904.285} C_VEL
LIN {X 0,Y 379.567,Z 434.8,A -85,B 0,C 180,E1 -17905.753,E2 -17905.753} C_VEL
LIN {X 0,Y 380.815,Z 435.243,A -85,B 0,C 180,E1 -17907.343,E2 -17907.343} C_VEL
LIN {X 0,Y 381.48,Z 435.643,A -85,B 0,C 180,E1 -17908.944,E2 -17908.944} C_VEL
LIN {X 0,Y 381.624,Z 435.577,A -85,B 0,C 180,E1 -17910,E2 -17910} C_VEL
LIN {X 0,Y 381.313,Z 435.52,A -85,B 0,C 180,E1 -17911.584,E2 -17911.584} C_VEL
LIN {X 0,Y 380.223,Z 434.937,A -85,B 0,C 180,E1 -17913.517,E2 -17913.517} C_VEL
LIN {X 0,Y 378.119,Z 434.211,A -85,B 0,C 180,E1 -17915.576,E2 -17915.576} C_VEL
LIN {X 0,Y 375.244,Z 432.718,A -85,B 0,C 180,E1 -17917.533,E2 -17917.533} C_VEL
LIN {X 0,Y 371.851,Z 430.567,A -85,B 0,C 180,E1 -17919.344,E2 -17919.344} C_VEL
LIN {X 0,Y 367.961,Z 427.425,A -85,B 0,C 180,E1 -17921.09,E2 -17921.09} C_VEL
LIN {X 0,Y 365.688,Z 425.801,A -85,B 0,C 180,E1 -17921.978,E2 -17921.978} C_VEL
LIN {X 0,Y 360.935,Z 422.934,A -85,B 0,C 180,E1 -17923.619,E2 -17923.619} C_VEL
LIN {X 0,Y 354.984,Z 418.367,A -85,B 0,C 180,E1 -17925.442,E2 -17925.442} C_VEL
LIN {X 0,Y 349.159,Z 414.144,A -85,B 0,C 180,E1 -17927.007,E2 -17927.007} C_VEL
LIN {X 0,Y 343.182,Z 409.292,A -85,B 0,C 180,E1 -17928.482,E2 -17928.482} C_VEL
LIN {X 0,Y 335.487,Z 403.191,A -85,B 0,C 180,E1 -17930.193,E2 -17930.193} C_VEL
LIN {X 0,Y 326.866,Z 395.85,A -85,B 0,C 180,E1 -17931.919,E2 -17931.919} C_VEL
LIN {X 0,Y 318.478,Z 388.196,A -85,B 0,C 180,E1 -17933.404,E2 -17933.404} C_VEL
LIN {X 0,Y 309.567,Z 379.809,A -85,B 0,C 180,E1 -17934.757,E2 -17934.757} C_VEL
LIN {X 0,Y 300.816,Z 370.822,A -85,B 0,C 180,E1 -17935.908,E2 -17935.908} C_VEL
LIN {X 0,Y 291.112,Z 360.01,A -85,B 0,C 180,E1 -17937.141,E2 -17937.141} C_VEL
LIN {X 0,Y 282.952,Z 348.523,A -85,B 0,C 180,E1 -17938.323,E2 -17938.323} C_VEL
LIN {X 0,Y 275.735,Z 335.361,A -85,B 0,C 180,E1 -17939.527,E2 -17939.527} C_VEL
LIN {X 0,Y 271.299,Z 327.281,A -85,B 0,C 180,E1 -17940.306,E2 -17940.306} C_VEL
LIN {X 0,Y 270.367,Z 325.031,A -85,B 0,C 180,E1 -17940.562,E2 -17940.562} C_VEL
LIN {X 0,Y 270.202,Z 324.376,A -85,B 0,C 180,E1 -17940.872,E2 -17940.872} C_VEL
LIN {X 0,Y 270.21,Z 324.289,A -85,B 0,C 180,E1 -17944.903,E2 -17944.903} C_VEL
LIN {X 0,Y 270.217,Z 324.32,A -85,B 0,C 180,E1 -17948.717,E2 -17948.717} C_VEL
LIN {X 0,Y 270.183,Z 324.279,A -85,B 0,C 180,E1 -17953.254,E2 -17953.254} C_VEL
LIN {X 0,Y 270.216,Z 324.322,A -85,B 0,C 180,E1 -17957.452,E2 -17957.452} C_VEL
LIN {X 0,Y 270.239,Z 324.321,A -85,B 0,C 180,E1 -17961.381,E2 -17961.381} C_VEL
LIN {X 0,Y 270.209,Z 324.304,A -85,B 0,C 180,E1 -17965.097,E2 -17965.097} C_VEL
LIN {X 0,Y 270.194,Z 324.331,A -85,B 0,C 180,E1 -17969.131,E2 -17969.131} C_VEL
LIN {X 0,Y 270.257,Z 324.292,A -85,B 0,C 180,E1 -17972.146,E2 -17972.146} C_VEL
LIN {X 0,Y 270.27,Z 324.316,A -85,B 0,C 180,E1 -17975.52,E2 -17975.52} C_VEL
LIN {X 0,Y 270.295,Z 324.282,A -85,B 0,C 180,E1 -17980.245,E2 -17980.245} C_VEL
LIN {X 0,Y 270.39,Z 324.305,A -85,B 0,C 180,E1 -17984.936,E2 -17984.936} C_VEL
LIN {X 0,Y 270.406,Z 324.26,A -85,B 0,C 180,E1 -17989.518,E2 -17989.518} C_VEL
LIN {X 0,Y 270.592,Z 324.264,A -85,B 0,C 180,E1 -17992.539,E2 -17992.539} C_VEL
LIN {X 0,Y 270.78,Z 324.218,A -85,B 0,C 180,E1 -17998.514,E2 -17998.514} C_VEL
LIN {X 0,Y 270.781,Z 324.227,A -85,B 0,C 180,E1 -18001.488,E2 -18001.488} C_VEL
LIN {X 0,Y 270.593,Z 324.256,A -85,B 0,C 180,E1 -18007.462,E2 -18007.462} C_VEL
LIN {X 0,Y 270.407,Z 324.263,A -85,B 0,C 180,E1 -18010.483,E2 -18010.483} C_VEL
LIN {X 0,Y 270.391,Z 324.297,A -85,B 0,C 180,E1 -18015.066,E2 -18015.066} C_VEL
LIN {X 0,Y 270.295,Z 324.285,A -85,B 0,C 180,E1 -18019.757,E2 -18019.757} C_VEL
LIN {X 0,Y 270.234,Z 324.311,A -85,B 0,C 180,E1 -18024.59,E2 -18024.59} C_VEL
LIN {X 0,Y 270.266,Z 324.295,A -85,B 0,C 180,E1 -18027.91,E2 -18027.91} C_VEL
LIN {X 0,Y 270.181,Z 324.328,A -85,B 0,C 180,E1 -18031.349,E2 -18031.349} C_VEL
LIN {X 0,Y 270.176,Z 324.312,A -85,B 0,C 180,E1 -18032.762,E2 -18032.762} C_VEL
LIN {X 0,Y 269.563,Z 324.389,A -85,B 0,C 180,E1 -18034.007,E2 -18034.007} C_VEL
LIN {X 0,Y 266.727,Z 324.753,A -85,B 0,C 180,E1 -18036.036,E2 -18036.036} C_VEL
LIN {X 0,Y 264.276,Z 325.066,A -85,B 0,C 180,E1 -18037.685,E2 -18037.685} C_VEL
LIN {X 0,Y 263.205,Z 325.188,A -85,B 0,C 180,E1 -18038.964,E2 -18038.964} C_VEL
LIN {X 0,Y 263.11,Z 325.196,A -85,B 0,C 180,E1 -18039.397,E2 -18039.397} C_VEL
LIN {X 0,Y 263.122,Z 325.208,A -85,B 0,C 180,E1 -18041.895,E2 -18041.895} C_VEL
LIN {X 0,Y 263.098,Z 325.215,A -85,B 0,C 180,E1 -18046.158,E2 -18046.158} C_VEL
LIN {X 0,Y 263.089,Z 325.189,A -85,B 0,C 180,E1 -18050.778,E2 -18050.778} C_VEL
LIN {X 0,Y 263.168,Z 325.366,A -85,B 0,C 180,E1 -18051.633,E2 -18051.633} C_VEL
LIN {X 0,Y 264.8,Z 332.674,A -85,B 0,C 180,E1 -18055.364,E2 -18055.364} C_VEL
LIN {X 0,Y 266.302,Z 340.263,A -85,B 0,C 180,E1 -18058.982,E2 -18058.982} C_VEL
LIN {X 0,Y 267.662,Z 343.703,A -85,B 0,C 180,E1 -18059.352,E2 -18059.352} C_VEL
LIN {X 0,Y 272.681,Z 355.785,A -85,B 0,C 180,E1 -18060.329,E2 -18060.329} C_VEL
LIN {X 0,Y 277.171,Z 377.937,A -85,B 0,C 180,E1 -18061.493,E2 -18061.493} C_VEL
LIN {X 0,Y 279.183,Z 390.912,A -85,B 0,C 180,E1 -18062.085,E2 -18062.085} C_VEL
LIN {X 0,Y 277.475,Z 446.667,A -85,B 0,C 180,E1 -18063.538,E2 -18063.538} C_VEL
LIN {X 0,Y 276.704,Z 456.96,A -85,B 0,C 180,E1 -18063.965,E2 -18063.965} C_VEL
LIN {X 0,Y 275.702,Z 466.469,A -85,B 0,C 180,E1 -18064.523,E2 -18064.523} C_VEL
LIN {X 0,Y 274.55,Z 475.54,A -85,B 0,C 180,E1 -18065.218,E2 -18065.218} C_VEL
LIN {X 0,Y 273.248,Z 484.671,A -85,B 0,C 180,E1 -18066.104,E2 -18066.104} C_VEL
LIN {X 0,Y 271.701,Z 493.663,A -85,B 0,C 180,E1 -18067.17,E2 -18067.17} C_VEL
LIN {X 0,Y 270.082,Z 502.388,A -85,B 0,C 180,E1 -18068.436,E2 -18068.436} C_VEL
LIN {X 0,Y 268.581,Z 509.779,A -85,B 0,C 180,E1 -18069.714,E2 -18069.714} C_VEL
LIN {X 0,Y 266.89,Z 518.059,A -85,B 0,C 180,E1 -18071.441,E2 -18071.441} C_VEL
LIN {X 0,Y 265.931,Z 523.203,A -85,B 0,C 180,E1 -18072.704,E2 -18072.704} C_VEL
LIN {X 0,Y 264.532,Z 529.74,A -85,B 0,C 180,E1 -18074.593,E2 -18074.593} C_VEL
LIN {X 0,Y 263.516,Z 534.24,A -85,B 0,C 180,E1 -18076.112,E2 -18076.112} C_VEL
LIN {X 0,Y 262.421,Z 539.733,A -85,B 0,C 180,E1 -18078.413,E2 -18078.413} C_VEL
LIN {X 0,Y 261.702,Z 544.061,A -85,B 0,C 180,E1 -18080.728,E2 -18080.728} C_VEL
LIN {X 0,Y 261.354,Z 546.429,A -85,B 0,C 180,E1 -18082.273,E2 -18082.273} C_VEL
LIN {X 0,Y 261.087,Z 549.235,A -85,B 0,C 180,E1 -18084.865,E2 -18084.865} C_VEL
LIN {X 0,Y 261.054,Z 550.683,A -85,B 0,C 180,E1 -18086.914,E2 -18086.914} C_VEL
LIN {X 0,Y 261.088,Z 551.275,A -85,B 0,C 180,E1 -18088.458,E2 -18088.458} C_VEL
LIN {X 0,Y 261.088,Z 551.275,A -85,B 0,C 180,E1 -18091.542,E2 -18091.542} C_VEL
LIN {X 0,Y 261.052,Z 550.683,A -85,B 0,C 180,E1 -18093.086,E2 -18093.086} C_VEL
LIN {X 0,Y 261.151,Z 548.231,A -85,B 0,C 180,E1 -18096.18,E2 -18096.18} C_VEL
LIN {X 0,Y 261.518,Z 545.279,A -85,B 0,C 180,E1 -18098.5,E2 -18098.5} C_VEL
LIN {X 0,Y 262.136,Z 541.287,A -85,B 0,C 180,E1 -18100.817,E2 -18100.817} C_VEL
LIN {X 0,Y 263.09,Z 536.155,A -85,B 0,C 180,E1 -18103.124,E2 -18103.124} C_VEL
LIN {X 0,Y 264.247,Z 530.894,A -85,B 0,C 180,E1 -18105.029,E2 -18105.029} C_VEL
LIN {X 0,Y 265.594,Z 524.578,A -85,B 0,C 180,E1 -18106.922,E2 -18106.922} C_VEL
LIN {X 0,Y 266.864,Z 518.627,A -85,B 0,C 180,E1 -18108.422,E2 -18108.422} C_VEL
LIN {X 0,Y 268.224,Z 511.699,A -85,B 0,C 180,E1 -18109.915,E2 -18109.915} C_VEL
LIN {X 0,Y 269.842,Z 503.522,A -85,B 0,C 180,E1 -18111.384,E2 -18111.384} C_VEL
LIN {X 0,Y 271.481,Z 495.015,A -85,B 0,C 180,E1 -18112.648,E2 -18112.648} C_VEL
LIN {X 0,Y 272.997,Z 486.303,A -85,B 0,C 180,E1 -18113.718,E2 -18113.718} C_VEL
LIN {X 0,Y 274.388,Z 476.546,A -85,B 0,C 180,E1 -18114.696,E2 -18114.696} C_VEL
LIN {X 0,Y 275.562,Z 467.757,A -85,B 0,C 180,E1 -18115.39,E2 -18115.39} C_VEL
LIN {X 0,Y 276.59,Z 457.833,A -85,B 0,C 180,E1 -18115.996,E2 -18115.996} C_VEL
LIN {X 0,Y 277.373,Z 447.985,A -85,B 0,C 180,E1 -18116.422,E2 -18116.422} C_VEL
LIN {X 0,Y 278.256,Z 422.479,A -85,B 0,C 180,E1 -18117.117,E2 -18117.117} C_VEL
LIN {X 0,Y 279.112,Z 389.627,A -85,B 0,C 180,E1 -18117.959,E2 -18117.959} C_VEL
LIN {X 0,Y 275.187,Z 367.736,A -85,B 0,C 180,E1 -18119.028,E2 -18119.028} C_VEL
LIN {X 0,Y 272.223,Z 354.326,A -85,B 0,C 180,E1 -18119.769,E2 -18119.769} C_VEL
LIN {X 0,Y 266.397,Z 340.704,A -85,B 0,C 180,E1 -18120.932,E2 -18120.932} C_VEL
LIN {X 0,Y 266.133,Z 339.516,A -85,B 0,C 180,E1 -18121.295,E2 -18121.295} C_VEL
LIN {X 0,Y 264.588,Z 331.748,A -85,B 0,C 180,E1 -18125.097,E2 -18125.097} C_VEL
LIN {X 0,Y 263.158,Z 325.251,A -85,B 0,C 180,E1 -18128.488,E2 -18128.488} C_VEL
LIN {X 0,Y 263.074,Z 325.192,A -85,B 0,C 180,E1 -18131.902,E2 -18131.902} C_VEL
LIN {X 0,Y 263.104,Z 325.203,A -85,B 0,C 180,E1 -18136.154,E2 -18136.154} C_VEL
LIN {X 0,Y 263.104,Z 325.196,A -85,B 0,C 180,E1 -18140.126,E2 -18140.126} C_VEL
LIN {X 0,Y 263.16,Z 325.197,A -85,B 0,C 180,E1 -18144.017,E2 -18144.017} C_VEL
LIN {X 0,Y 263.13,Z 325.196,A -85,B 0,C 180,E1 -18147.71,E2 -18147.71} C_VEL
LIN {X 0,Y 263.192,Z 325.179,A -85,B 0,C 180,E1 -18151.784,E2 -18151.784} C_VEL
LIN {X 0,Y 263.197,Z 325.186,A -85,B 0,C 180,E1 -18155.211,E2 -18155.211} C_VEL
LIN {X 0,Y 263.258,Z 325.168,A -85,B 0,C 180,E1 -18159.692,E2 -18159.692} C_VEL
LIN {X 0,Y 263.34,Z 325.174,A -85,B 0,C 180,E1 -18164.521,E2 -18164.521} C_VEL
LIN {X 0,Y 263.35,Z 325.144,A -85,B 0,C 180,E1 -18169.233,E2 -18169.233} C_VEL
LIN {X 0,Y 263.552,Z 325.127,A -85,B 0,C 180,E1 -18172.337,E2 -18172.337} C_VEL
LIN {X 0,Y 263.745,Z 325.103,A -85,B 0,C 180,E1 -18178.472,E2 -18178.472} C_VEL
LIN {X 0,Y 263.744,Z 325.094,A -85,B 0,C 180,E1 -18181.526,E2 -18181.526} C_VEL
LIN {X 0,Y 263.551,Z 325.139,A -85,B 0,C 180,E1 -18187.661,E2 -18187.661} C_VEL
LIN {X 0,Y 263.348,Z 325.14,A -85,B 0,C 180,E1 -18190.766,E2 -18190.766} C_VEL
LIN {X 0,Y 263.338,Z 325.18,A -85,B 0,C 180,E1 -18195.478,E2 -18195.478} C_VEL
LIN {X 0,Y 263.257,Z 325.162,A -85,B 0,C 180,E1 -18200.306,E2 -18200.306} C_VEL
LIN {X 0,Y 263.202,Z 325.188,A -85,B 0,C 180,E1 -18205.291,E2 -18205.291} C_VEL
LIN {X 0,Y 263.16,Z 325.183,A -85,B 0,C 180,E1 -18208.731,E2 -18208.731} C_VEL
LIN {X 0,Y 263.127,Z 325.205,A -85,B 0,C 180,E1 -18212.288,E2 -18212.288} C_VEL
LIN {X 0,Y 263.183,Z 325.189,A -85,B 0,C 180,E1 -18215.978,E2 -18215.978} C_VEL
LIN {X 0,Y 263.153,Z 325.19,A -85,B 0,C 180,E1 -18219.863,E2 -18219.863} C_VEL
LIN {X 0,Y 263.139,Z 325.206,A -85,B 0,C 180,E1 -18223.979,E2 -18223.979} C_VEL
LIN {X 0,Y 263.125,Z 325.15,A -85,B 0,C 180,E1 -18228.405,E2 -18228.405} C_VEL
LIN {X 0,Y 263.163,Z 325.207,A -85,B 0,C 180,E1 -18232.105,E2 -18232.105} C_VEL
LIN {X 0,Y 263.179,Z 325.165,A -85,B 0,C 180,E1 -18235.89,E2 -18235.89} C_VEL
LIN {X 0,Y 263.169,Z 325.412,A -85,B 0,C 180,E1 -18238.397,E2 -18238.397} C_VEL
LIN {X 0,Y 263.399,Z 326.396,A -85,B 0,C 180,E1 -18238.628,E2 -18238.628} C_VEL
LIN {X 0,Y 271.761,Z 341.955,A -85,B 0,C 180,E1 -18240.191,E2 -18240.191} C_VEL
LIN {X 0,Y 277.976,Z 353.13,A -85,B 0,C 180,E1 -18241.251,E2 -18241.251} C_VEL
LIN {X 0,Y 286.581,Z 365.26,A -85,B 0,C 180,E1 -18242.535,E2 -18242.535} C_VEL
LIN {X 0,Y 298.695,Z 378.675,A -85,B 0,C 180,E1 -18244.098,E2 -18244.098} C_VEL
LIN {X 0,Y 308.559,Z 388.263,A -85,B 0,C 180,E1 -18245.357,E2 -18245.357} C_VEL
LIN {X 0,Y 317.168,Z 396.09,A -85,B 0,C 180,E1 -18246.644,E2 -18246.644} C_VEL
LIN {X 0,Y 325.044,Z 403.042,A -85,B 0,C 180,E1 -18248.004,E2 -18248.004} C_VEL
LIN {X 0,Y 332.832,Z 409.602,A -85,B 0,C 180,E1 -18249.521,E2 -18249.521} C_VEL
LIN {X 0,Y 341.236,Z 416.13,A -85,B 0,C 180,E1 -18251.332,E2 -18251.332} C_VEL
LIN {X 0,Y 347.504,Z 421.066,A -85,B 0,C 180,E1 -18252.854,E2 -18252.854} C_VEL
LIN {X 0,Y 352.785,Z 424.836,A -85,B 0,C 180,E1 -18254.248,E2 -18254.248} C_VEL
LIN {X 0,Y 357.584,Z 428.522,A -85,B 0,C 180,E1 -18255.658,E2 -18255.658} C_VEL
LIN {X 0,Y 362.643,Z 431.81,A -85,B 0,C 180,E1 -18257.285,E2 -18257.285} C_VEL
LIN {X 0,Y 366.023,Z 433.796,A -85,B 0,C 180,E1 -18258.506,E2 -18258.506} C_VEL
LIN {X 0,Y 370.011,Z 437.038,A -85,B 0,C 180,E1 -18260.217,E2 -18260.217} C_VEL
LIN {X 0,Y 373.567,Z 439.361,A -85,B 0,C 180,E1 -18262.024,E2 -18262.024} C_VEL
LIN {X 0,Y 376.284,Z 440.836,A -85,B 0,C 180,E1 -18263.721,E2 -18263.721} C_VEL
LIN {X 0,Y 378.681,Z 441.843,A -85,B 0,C 180,E1 -18265.743,E2 -18265.743} C_VEL
LIN {X 0,Y 379.929,Z 442.268,A -85,B 0,C 180,E1 -18267.3,E2 -18267.3} C_VEL
LIN {X 0,Y 380.613,Z 442.689,A -85,B 0,C 180,E1 -18268.942,E2 -18268.942} C_VEL
LIN {X 0,Y 380.758,Z 442.623,A -85,B 0,C 180,E1 -18270,E2 -18270} C_VEL
LIN {X 0,Y 380.444,Z 442.566,A -85,B 0,C 180,E1 -18271.588,E2 -18271.588} C_VEL
LIN {X 0,Y 379.6,Z 442.063,A -85,B 0,C 180,E1 -18273.184,E2 -18273.184} C_VEL
LIN {X 0,Y 377.821,Z 441.523,A -85,B 0,C 180,E1 -18275.066,E2 -18275.066} C_VEL
LIN {X 0,Y 375.25,Z 440.304,A -85,B 0,C 180,E1 -18276.967,E2 -18276.967} C_VEL
LIN {X 0,Y 371.736,Z 438.237,A -85,B 0,C 180,E1 -18278.955,E2 -18278.955} C_VEL
LIN {X 0,Y 368.052,Z 435.54,A -85,B 0,C 180,E1 -18280.654,E2 -18280.654} C_VEL
LIN {X 0,Y 364.634,Z 432.867,A -85,B 0,C 180,E1 -18282.014,E2 -18282.014} C_VEL
LIN {X 0,Y 359.519,Z 429.863,A -85,B 0,C 180,E1 -18283.755,E2 -18283.755} C_VEL
LIN {X 0,Y 353.673,Z 425.58,A -85,B 0,C 180,E1 -18285.504,E2 -18285.504} C_VEL
LIN {X 0,Y 349.314,Z 422.272,A -85,B 0,C 180,E1 -18286.692,E2 -18286.692} C_VEL
LIN {X 0,Y 343.081,Z 417.725,A -85,B 0,C 180,E1 -18288.224,E2 -18288.224} C_VEL
LIN {X 0,Y 337.556,Z 413.268,A -85,B 0,C 180,E1 -18289.487,E2 -18289.487} C_VEL
LIN {X 0,Y 330.474,Z 407.531,A -85,B 0,C 180,E1 -18290.965,E2 -18290.965} C_VEL
LIN {X 0,Y 321.984,Z 400.395,A -85,B 0,C 180,E1 -18292.55,E2 -18292.55} C_VEL
LIN {X 0,Y 313.092,Z 392.428,A -85,B 0,C 180,E1 -18293.994,E2 -18293.994} C_VEL
LIN {X 0,Y 304.444,Z 384.311,A -85,B 0,C 180,E1 -18295.193,E2 -18295.193} C_VEL
LIN {X 0,Y 292.366,Z 371.984,A -85,B 0,C 180,E1 -18296.691,E2 -18296.691} C_VEL
LIN {X 0,Y 284.26,Z 362.165,A -85,B 0,C 180,E1 -18297.797,E2 -18297.797} C_VEL
LIN {X 0,Y 276.971,Z 351.495,A -85,B 0,C 180,E1 -18298.911,E2 -18298.911} C_VEL
LIN {X 0,Y 264.623,Z 328.757,A -85,B 0,C 180,E1 -18301.116,E2 -18301.116} C_VEL
LIN {X 0,Y 263.299,Z 326.061,A -85,B 0,C 180,E1 -18301.427,E2 -18301.427} C_VEL
LIN {X 0,Y 263.124,Z 325.266,A -85,B 0,C 180,E1 -18301.787,E2 -18301.787} C_VEL
LIN {X 0,Y 263.168,Z 325.166,A -85,B 0,C 180,E1 -18304.122,E2 -18304.122} C_VEL
LIN {X 0,Y 263.163,Z 325.207,A -85,B 0,C 180,E1 -18307.895,E2 -18307.895} C_VEL
LIN {X 0,Y 263.126,Z 325.149,A -85,B 0,C 180,E1 -18311.892,E2 -18311.892} C_VEL
LIN {X 0,Y 263.141,Z 325.207,A -85,B 0,C 180,E1 -18316.146,E2 -18316.146} C_VEL
LIN {X 0,Y 263.153,Z 325.19,A -85,B 0,C 180,E1 -18320.137,E2 -18320.137} C_VEL
LIN {X 0,Y 263.183,Z 325.189,A -85,B 0,C 180,E1 -18324.022,E2 -18324.022} C_VEL
LIN {X 0,Y 263.127,Z 325.205,A -85,B 0,C 180,E1 -18327.712,E2 -18327.712} C_VEL
LIN {X 0,Y 263.19,Z 325.174,A -85,B 0,C 180,E1 -18331.785,E2 -18331.785} C_VEL
LIN {X 0,Y 263.219,Z 325.19,A -85,B 0,C 180,E1 -18335.201,E2 -18335.201} C_VEL
LIN {X 0,Y 263.257,Z 325.162,A -85,B 0,C 180,E1 -18339.694,E2 -18339.694} C_VEL
LIN {X 0,Y 263.338,Z 325.18,A -85,B 0,C 180,E1 -18344.522,E2 -18344.522} C_VEL
LIN {X 0,Y 263.348,Z 325.14,A -85,B 0,C 180,E1 -18349.234,E2 -18349.234} C_VEL
LIN {X 0,Y 263.551,Z 325.139,A -85,B 0,C 180,E1 -18352.339,E2 -18352.339} C_VEL
LIN {X 0,Y 263.744,Z 325.094,A -85,B 0,C 180,E1 -18358.474,E2 -18358.474} C_VEL
LIN {X 0,Y 263.745,Z 325.103,A -85,B 0,C 180,E1 -18361.528,E2 -18361.528} C_VEL
LIN {X 0,Y 263.552,Z 325.127,A -85,B 0,C 180,E1 -18367.663,E2 -18367.663} C_VEL
LIN {X 0,Y 263.35,Z 325.144,A -85,B 0,C 180,E1 -18370.767,E2 -18370.767} C_VEL
LIN {X 0,Y 263.34,Z 325.174,A -85,B 0,C 180,E1 -18375.479,E2 -18375.479} C_VEL
LIN {X 0,Y 263.258,Z 325.168,A -85,B 0,C 180,E1 -18380.308,E2 -18380.308} C_VEL
LIN {X 0,Y 263.188,Z 325.18,A -85,B 0,C 180,E1 -18385.294,E2 -18385.294} C_VEL
LIN {X 0,Y 263.162,Z 325.189,A -85,B 0,C 180,E1 -18388.733,E2 -18388.733} C_VEL
LIN {X 0,Y 263.109,Z 325.193,A -85,B 0,C 180,E1 -18392.754,E2 -18392.754} C_VEL
LIN {X 0,Y 263.179,Z 325.203,A -85,B 0,C 180,E1 -18396.764,E2 -18396.764} C_VEL
LIN {X 0,Y 263.11,Z 325.196,A -85,B 0,C 180,E1 -18399.397,E2 -18399.397} C_VEL
LIN {X 0,Y 262.417,Z 325.285,A -85,B 0,C 180,E1 -18400.675,E2 -18400.675} C_VEL
LIN {X 0,Y 259.545,Z 325.654,A -85,B 0,C 180,E1 -18402.757,E2 -18402.757} C_VEL
LIN {X 0,Y 257.128,Z 325.953,A -85,B 0,C 180,E1 -18404.451,E2 -18404.451} C_VEL
LIN {X 0,Y 256.101,Z 326.082,A -85,B 0,C 180,E1 -18405.764,E2 -18405.764} C_VEL
LIN {X 0,Y 256.023,Z 326.091,A -85,B 0,C 180,E1 -18406.209,E2 -18406.209} C_VEL
LIN {X 0,Y 256.062,Z 326.148,A -85,B 0,C 180,E1 -18410.857,E2 -18410.857} C_VEL
LIN {X 0,Y 257.474,Z 332.108,A -85,B 0,C 180,E1 -18414.067,E2 -18414.067} C_VEL
LIN {X 0,Y 259.058,Z 339.971,A -85,B 0,C 180,E1 -18417.995,E2 -18417.995} C_VEL
LIN {X 0,Y 259.754,Z 342.167,A -85,B 0,C 180,E1 -18418.272,E2 -18418.272} C_VEL
LIN {X 0,Y 264.747,Z 353.27,A -85,B 0,C 180,E1 -18419.276,E2 -18419.276} C_VEL
LIN {X 0,Y 266.901,Z 358.787,A -85,B 0,C 180,E1 -18419.716,E2 -18419.716} C_VEL
LIN {X 0,Y 271.424,Z 381.98,A -85,B 0,C 180,E1 -18420.957,E2 -18420.957} C_VEL
LIN {X 0,Y 272.91,Z 391.68,A -85,B 0,C 180,E1 -18421.413,E2 -18421.413} C_VEL
LIN {X 0,Y 271.144,Z 446.596,A -85,B 0,C 180,E1 -18422.875,E2 -18422.875} C_VEL
LIN {X 0,Y 270.325,Z 456.804,A -85,B 0,C 180,E1 -18423.305,E2 -18423.305} C_VEL
LIN {X 0,Y 269.311,Z 466.276,A -85,B 0,C 180,E1 -18423.873,E2 -18423.873} C_VEL
LIN {X 0,Y 267.99,Z 476.353,A -85,B 0,C 180,E1 -18424.673,E2 -18424.673} C_VEL
LIN {X 0,Y 266.748,Z 484.477,A -85,B 0,C 180,E1 -18425.484,E2 -18425.484} C_VEL
LIN {X 0,Y 265.168,Z 493.469,A -85,B 0,C 180,E1 -18426.575,E2 -18426.575} C_VEL
LIN {X 0,Y 263.49,Z 502.194,A -85,B 0,C 180,E1 -18427.868,E2 -18427.868} C_VEL
LIN {X 0,Y 261.92,Z 509.585,A -85,B 0,C 180,E1 -18429.175,E2 -18429.175} C_VEL
LIN {X 0,Y 260.382,Z 516.803,A -85,B 0,C 180,E1 -18430.693,E2 -18430.693} C_VEL
LIN {X 0,Y 259.117,Z 523.159,A -85,B 0,C 180,E1 -18432.279,E2 -18432.279} C_VEL
LIN {X 0,Y 257.661,Z 529.545,A -85,B 0,C 180,E1 -18434.172,E2 -18434.172} C_VEL
LIN {X 0,Y 256.623,Z 534.046,A -85,B 0,C 180,E1 -18435.731,E2 -18435.731} C_VEL
LIN {X 0,Y 255.44,Z 539.538,A -85,B 0,C 180,E1 -18438.092,E2 -18438.092} C_VEL
LIN {X 0,Y 254.655,Z 543.866,A -85,B 0,C 180,E1 -18440.469,E2 -18440.469} C_VEL
LIN {X 0,Y 254.314,Z 546.235,A -85,B 0,C 180,E1 -18442.058,E2 -18442.058} C_VEL
LIN {X 0,Y 253.993,Z 549.221,A -85,B 0,C 180,E1 -18444.961,E2 -18444.961} C_VEL
LIN {X 0,Y 253.954,Z 550.489,A -85,B 0,C 180,E1 -18446.827,E2 -18446.827} C_VEL
LIN {X 0,Y 253.995,Z 551.081,A -85,B 0,C 180,E1 -18448.414,E2 -18448.414} C_VEL
LIN {X 0,Y 254.046,Z 551.238,A -85,B 0,C 180,E1 -18450,E2 -18450} C_VEL
LIN {X 0,Y 253.995,Z 551.081,A -85,B 0,C 180,E1 -18451.586,E2 -18451.586} C_VEL
LIN {X 0,Y 253.952,Z 550.489,A -85,B 0,C 180,E1 -18453.173,E2 -18453.173} C_VEL
LIN {X 0,Y 254.063,Z 548.036,A -85,B 0,C 180,E1 -18456.353,E2 -18456.353} C_VEL
LIN {X 0,Y 254.475,Z 545.084,A -85,B 0,C 180,E1 -18458.737,E2 -18458.737} C_VEL
LIN {X 0,Y 255.128,Z 541.092,A -85,B 0,C 180,E1 -18461.118,E2 -18461.118} C_VEL
LIN {X 0,Y 256.138,Z 535.96,A -85,B 0,C 180,E1 -18463.487,E2 -18463.487} C_VEL
LIN {X 0,Y 257.381,Z 530.7,A -85,B 0,C 180,E1 -18465.44,E2 -18465.44} C_VEL
LIN {X 0,Y 258.798,Z 524.383,A -85,B 0,C 180,E1 -18467.38,E2 -18467.38} C_VEL
LIN {X 0,Y 260.154,Z 518.103,A -85,B 0,C 180,E1 -18468.998,E2 -18468.998} C_VEL
LIN {X 0,Y 261.524,Z 511.504,A -85,B 0,C 180,E1 -18470.447,E2 -18470.447} C_VEL
LIN {X 0,Y 263.246,Z 503.328,A -85,B 0,C 180,E1 -18471.947,E2 -18471.947} C_VEL
LIN {X 0,Y 264.918,Z 494.82,A -85,B 0,C 180,E1 -18473.242,E2 -18473.242} C_VEL
LIN {X 0,Y 266.506,Z 486.109,A -85,B 0,C 180,E1 -18474.333,E2 -18474.333} C_VEL
LIN {X 0,Y 267.935,Z 476.351,A -85,B 0,C 180,E1 -18475.333,E2 -18475.333} C_VEL
LIN {X 0,Y 269.328,Z 466.276,A -85,B 0,C 180,E1 -18476.125,E2 -18476.125} C_VEL
LIN {X 0,Y 270.313,Z 456.8,A -85,B 0,C 180,E1 -18476.696,E2 -18476.696} C_VEL
LIN {X 0,Y 271.095,Z 446.569,A -85,B 0,C 180,E1 -18477.131,E2 -18477.131} C_VEL
LIN {X 0,Y 272.929,Z 391.277,A -85,B 0,C 180,E1 -18478.597,E2 -18478.597} C_VEL
LIN {X 0,Y 268.923,Z 368.638,A -85,B 0,C 180,E1 -18479.738,E2 -18479.738} C_VEL
LIN {X 0,Y 266.357,Z 357.105,A -85,B 0,C 180,E1 -18480.403,E2 -18480.403} C_VEL
LIN {X 0,Y 259.138,Z 340.333,A -85,B 0,C 180,E1 -18481.918,E2 -18481.918} C_VEL
LIN {X 0,Y 258.652,Z 337.985,A -85,B 0,C 180,E1 -18482.917,E2 -18482.917} C_VEL
LIN {X 0,Y 257.049,Z 330.104,A -85,B 0,C 180,E1 -18486.977,E2 -18486.977} C_VEL
LIN {X 0,Y 256.063,Z 326.161,A -85,B 0,C 180,E1 -18489.143,E2 -18489.143} C_VEL
LIN {X 0,Y 256.033,Z 326.093,A -85,B 0,C 180,E1 -18493.332,E2 -18493.332} C_VEL
LIN {X 0,Y 256.068,Z 326.089,A -85,B 0,C 180,E1 -18497.818,E2 -18497.818} C_VEL
LIN {X 0,Y 256.07,Z 326.074,A -85,B 0,C 180,E1 -18500.857,E2 -18500.857} C_VEL
LIN {X 0,Y 256.127,Z 326.081,A -85,B 0,C 180,E1 -18502.866,E2 -18502.866} C_VEL
LIN {X 0,Y 256.065,Z 326.066,A -85,B 0,C 180,E1 -18506.706,E2 -18506.706} C_VEL
LIN {X 0,Y 256.101,Z 326.08,A -85,B 0,C 180,E1 -18510.398,E2 -18510.398} C_VEL
LIN {X 0,Y 256.167,Z 326.056,A -85,B 0,C 180,E1 -18514.869,E2 -18514.869} C_VEL
LIN {X 0,Y 256.158,Z 326.059,A -85,B 0,C 180,E1 -18519.103,E2 -18519.103} C_VEL
LIN {X 0,Y 256.275,Z 326.048,A -85,B 0,C 180,E1 -18524.083,E2 -18524.083} C_VEL
LIN {X 0,Y 256.288,Z 326.05,A -85,B 0,C 180,E1 -18527.327,E2 -18527.327} C_VEL
LIN {X 0,Y 256.51,Z 326,A -85,B 0,C 180,E1 -18532.125,E2 -18532.125} C_VEL
LIN {X 0,Y 256.492,Z 326.028,A -85,B 0,C 180,E1 -18536.858,E2 -18536.858} C_VEL
LIN {X 0,Y 256.752,Z 325.957,A -85,B 0,C 180,E1 -18539.999,E2 -18539.999} C_VEL
LIN {X 0,Y 256.491,Z 326.021,A -85,B 0,C 180,E1 -18543.141,E2 -18543.141} C_VEL
LIN {X 0,Y 256.509,Z 326.01,A -85,B 0,C 180,E1 -18547.873,E2 -18547.873} C_VEL
LIN {X 0,Y 256.287,Z 326.048,A -85,B 0,C 180,E1 -18552.672,E2 -18552.672} C_VEL
LIN {X 0,Y 256.272,Z 326.054,A -85,B 0,C 180,E1 -18556.298,E2 -18556.298} C_VEL
LIN {X 0,Y 256.151,Z 326.058,A -85,B 0,C 180,E1 -18561.119,E2 -18561.119} C_VEL
LIN {X 0,Y 256.182,Z 326.064,A -85,B 0,C 180,E1 -18565.138,E2 -18565.138} C_VEL
LIN {X 0,Y 256.098,Z 326.074,A -85,B 0,C 180,E1 -18569.601,E2 -18569.601} C_VEL
LIN {X 0,Y 256.079,Z 326.07,A -85,B 0,C 180,E1 -18573.29,E2 -18573.29} C_VEL
LIN {X 0,Y 256.135,Z 326.082,A -85,B 0,C 180,E1 -18577.279,E2 -18577.279} C_VEL
LIN {X 0,Y 256.097,Z 326.067,A -85,B 0,C 180,E1 -18581.194,E2 -18581.194} C_VEL
LIN {X 0,Y 256.07,Z 326.08,A -85,B 0,C 180,E1 -18584.474,E2 -18584.474} C_VEL
LIN {X 0,Y 256.056,Z 326.032,A -85,B 0,C 180,E1 -18588.798,E2 -18588.798} C_VEL
LIN {X 0,Y 256.142,Z 326.069,A -85,B 0,C 180,E1 -18592.87,E2 -18592.87} C_VEL
LIN {X 0,Y 256.096,Z 326.11,A -85,B 0,C 180,E1 -18597.303,E2 -18597.303} C_VEL
LIN {X 0,Y 256.252,Z 326.975,A -85,B 0,C 180,E1 -18597.643,E2 -18597.643} C_VEL
LIN {X 0,Y 257.771,Z 329.858,A -85,B 0,C 180,E1 -18597.989,E2 -18597.989} C_VEL
LIN {X 0,Y 266.204,Z 345.404,A -85,B 0,C 180,E1 -18599.604,E2 -18599.604} C_VEL
LIN {X 0,Y 272.548,Z 357.037,A -85,B 0,C 180,E1 -18600.734,E2 -18600.734} C_VEL
LIN {X 0,Y 281.186,Z 369.374,A -85,B 0,C 180,E1 -18602.074,E2 -18602.074} C_VEL
LIN {X 0,Y 291.248,Z 380.774,A -85,B 0,C 180,E1 -18603.436,E2 -18603.436} C_VEL
LIN {X 0,Y 303.63,Z 393.115,A -85,B 0,C 180,E1 -18604.961,E2 -18604.961} C_VEL
LIN {X 0,Y 313.056,Z 401.539,A -85,B 0,C 180,E1 -18606.255,E2 -18606.255} C_VEL
LIN {X 0,Y 322.321,Z 409.53,A -85,B 0,C 180,E1 -18607.765,E2 -18607.765} C_VEL
LIN {X 0,Y 330.694,Z 416.398,A -85,B 0,C 180,E1 -18609.344,E2 -18609.344} C_VEL
LIN {X 0,Y 339.212,Z 422.933,A -85,B 0,C 180,E1 -18611.147,E2 -18611.147} C_VEL
LIN {X 0,Y 345.908,Z 428.035,A -85,B 0,C 180,E1 -18612.729,E2 -18612.729} C_VEL
LIN {X 0,Y 350.719,Z 431.388,A -85,B 0,C 180,E1 -18613.969,E2 -18613.969} C_VEL
LIN {X 0,Y 355.81,Z 435.246,A -85,B 0,C 180,E1 -18615.43,E2 -18615.43} C_VEL
LIN {X 0,Y 360.953,Z 438.554,A -85,B 0,C 180,E1 -18617.039,E2 -18617.039} C_VEL
LIN {X 0,Y 364.57,Z 440.718,A -85,B 0,C 180,E1 -18618.329,E2 -18618.329} C_VEL
LIN {X 0,Y 368.887,Z 444.062,A -85,B 0,C 180,E1 -18620.127,E2 -18620.127} C_VEL
LIN {X 0,Y 372.366,Z 446.278,A -85,B 0,C 180,E1 -18621.851,E2 -18621.851} C_VEL
LIN {X 0,Y 375.376,Z 447.886,A -85,B 0,C 180,E1 -18623.706,E2 -18623.706} C_VEL
LIN {X 0,Y 377.799,Z 448.86,A -85,B 0,C 180,E1 -18625.733,E2 -18625.733} C_VEL
LIN {X 0,Y 379.058,Z 449.316,A -85,B 0,C 180,E1 -18627.294,E2 -18627.294} C_VEL
LIN {X 0,Y 379.744,Z 449.734,A -85,B 0,C 180,E1 -18628.94,E2 -18628.94} C_VEL
LIN {X 0,Y 379.893,Z 449.67,A -85,B 0,C 180,E1 -18630,E2 -18630} C_VEL
LIN {X 0,Y 379.625,Z 449.632,A -85,B 0,C 180,E1 -18631.43,E2 -18631.43} C_VEL
LIN {X 0,Y 378.724,Z 449.103,A -85,B 0,C 180,E1 -18633.191,E2 -18633.191} C_VEL
LIN {X 0,Y 376.928,Z 448.57,A -85,B 0,C 180,E1 -18635.078,E2 -18635.078} C_VEL
LIN {X 0,Y 374.241,Z 447.316,A -85,B 0,C 180,E1 -18637.041,E2 -18637.041} C_VEL
LIN {X 0,Y 370.772,Z 445.321,A -85,B 0,C 180,E1 -18638.978,E2 -18638.978} C_VEL
LIN {X 0,Y 366.9,Z 442.592,A -85,B 0,C 180,E1 -18640.737,E2 -18640.737} C_VEL
LIN {X 0,Y 362.875,Z 439.571,A -85,B 0,C 180,E1 -18642.3,E2 -18642.3} C_VEL
LIN {X 0,Y 357.753,Z 436.595,A -85,B 0,C 180,E1 -18643.979,E2 -18643.979} C_VEL
LIN {X 0,Y 352.492,Z 432.807,A -85,B 0,C 180,E1 -18645.532,E2 -18645.532} C_VEL
LIN {X 0,Y 347.631,Z 429.193,A -85,B 0,C 180,E1 -18646.834,E2 -18646.834} C_VEL
LIN {X 0,Y 341.145,Z 424.538,A -85,B 0,C 180,E1 -18648.408,E2 -18648.408} C_VEL
LIN {X 0,Y 334.215,Z 419.098,A -85,B 0,C 180,E1 -18649.938,E2 -18649.938} C_VEL
LIN {X 0,Y 326.832,Z 413.136,A -85,B 0,C 180,E1 -18651.416,E2 -18651.416} C_VEL
LIN {X 0,Y 318.725,Z 406.485,A -85,B 0,C 180,E1 -18652.845,E2 -18652.845} C_VEL
LIN {X 0,Y 310.788,Z 399.58,A -85,B 0,C 180,E1 -18654.072,E2 -18654.072} C_VEL
LIN {X 0,Y 301.955,Z 391.557,A -85,B 0,C 180,E1 -18655.252,E2 -18655.252} C_VEL
LIN {X 0,Y 287.707,Z 377.071,A -85,B 0,C 180,E1 -18657.022,E2 -18657.022} C_VEL
LIN {X 0,Y 279.572,Z 367.197,A -85,B 0,C 180,E1 -18658.165,E2 -18658.165} C_VEL
LIN {X 0,Y 271.959,Z 356.077,A -85,B 0,C 180,E1 -18659.365,E2 -18659.365} C_VEL
LIN {X 0,Y 259.579,Z 333.133,A -85,B 0,C 180,E1 -18661.655,E2 -18661.655} C_VEL
LIN {X 0,Y 256.312,Z 327.149,A -85,B 0,C 180,E1 -18662.335,E2 -18662.335} C_VEL
LIN {X 0,Y 256.096,Z 326.153,A -85,B 0,C 180,E1 -18662.699,E2 -18662.699} C_VEL
LIN {X 0,Y 256.116,Z 326.044,A -85,B 0,C 180,E1 -18665.187,E2 -18665.187} C_VEL
LIN {X 0,Y 256.083,Z 326.066,A -85,B 0,C 180,E1 -18669.139,E2 -18669.139} C_VEL
LIN {X 0,Y 256.067,Z 326.035,A -85,B 0,C 180,E1 -18673.325,E2 -18673.325} C_VEL
LIN {X 0,Y 256.119,Z 326.074,A -85,B 0,C 180,E1 -18677.806,E2 -18677.806} C_VEL
LIN {X 0,Y 256.103,Z 326.077,A -85,B 0,C 180,E1 -18680.865,E2 -18680.865} C_VEL
LIN {X 0,Y 256.115,Z 326.06,A -85,B 0,C 180,E1 -18684.814,E2 -18684.814} C_VEL
LIN {X 0,Y 256.086,Z 326.086,A -85,B 0,C 180,E1 -18688.573,E2 -18688.573} C_VEL
LIN {X 0,Y 256.132,Z 326.05,A -85,B 0,C 180,E1 -18692.196,E2 -18692.196} C_VEL
LIN {X 0,Y 256.161,Z 326.076,A -85,B 0,C 180,E1 -18695.7,E2 -18695.7} C_VEL
LIN {X 0,Y 256.16,Z 326.054,A -85,B 0,C 180,E1 -18699.105,E2 -18699.105} C_VEL
LIN {X 0,Y 256.288,Z 326.057,A -85,B 0,C 180,E1 -18704.085,E2 -18704.085} C_VEL
LIN {X 0,Y 256.287,Z 326.048,A -85,B 0,C 180,E1 -18707.328,E2 -18707.328} C_VEL
LIN {X 0,Y 256.509,Z 326.01,A -85,B 0,C 180,E1 -18712.127,E2 -18712.127} C_VEL
LIN {X 0,Y 256.491,Z 326.021,A -85,B 0,C 180,E1 -18716.859,E2 -18716.859} C_VEL
LIN {X 0,Y 256.752,Z 325.957,A -85,B 0,C 180,E1 -18720.001,E2 -18720.001} C_VEL
LIN {X 0,Y 256.492,Z 326.028,A -85,B 0,C 180,E1 -18723.142,E2 -18723.142} C_VEL
LIN {X 0,Y 256.51,Z 326,A -85,B 0,C 180,E1 -18727.875,E2 -18727.875} C_VEL
LIN {X 0,Y 256.288,Z 326.05,A -85,B 0,C 180,E1 -18732.673,E2 -18732.673} C_VEL
LIN {X 0,Y 256.257,Z 326.045,A -85,B 0,C 180,E1 -18736.286,E2 -18736.286} C_VEL
LIN {X 0,Y 256.158,Z 326.059,A -85,B 0,C 180,E1 -18740.897,E2 -18740.897} C_VEL
LIN {X 0,Y 256.167,Z 326.056,A -85,B 0,C 180,E1 -18745.131,E2 -18745.131} C_VEL
LIN {X 0,Y 256.101,Z 326.08,A -85,B 0,C 180,E1 -18749.602,E2 -18749.602} C_VEL
LIN {X 0,Y 256.065,Z 326.066,A -85,B 0,C 180,E1 -18753.294,E2 -18753.294} C_VEL
LIN {X 0,Y 256.112,Z 326.083,A -85,B 0,C 180,E1 -18757.272,E2 -18757.272} C_VEL
LIN {X 0,Y 256.053,Z 326.082,A -85,B 0,C 180,E1 -18761.205,E2 -18761.205} C_VEL
LIN {X 0,Y 256.036,Z 326.088,A -85,B 0,C 180,E1 -18765.536,E2 -18765.536} C_VEL
LIN {X 0,Y 256.023,Z 326.091,A -85,B 0,C 180,E1 -18766.209,E2 -18766.209} C_VEL
LIN {X 0,Y 255.318,Z 326.184,A -85,B 0,C 180,E1 -18767.101,E2 -18767.101} C_VEL
LIN {X 0,Y 252.392,Z 326.516,A -85,B 0,C 180,E1 -18768.502,E2 -18768.502} C_VEL
LIN {X 0,Y 249.668,Z 327.08,A -85,B 0,C 180,E1 -18769.902,E2 -18769.902} C_VEL
LIN {X 0,Y 249.251,Z 328.127,A -85,B 0,C 180,E1 -18770.766,E2 -18770.766} C_VEL
LIN {X 0,Y 250.777,Z 334.677,A -85,B 0,C 180,E1 -18774.364,E2 -18774.364} C_VEL
LIN {X 0,Y 251.878,Z 339.986,A -85,B 0,C 180,E1 -18777.027,E2 -18777.027} C_VEL
LIN {X 0,Y 254.907,Z 346.912,A -85,B 0,C 180,E1 -18777.755,E2 -18777.755} C_VEL
LIN {X 0,Y 260.811,Z 360.516,A -85,B 0,C 180,E1 -18778.992,E2 -18778.992} C_VEL
LIN {X 0,Y 265.193,Z 382.793,A -85,B 0,C 180,E1 -18780.237,E2 -18780.237} C_VEL
LIN {X 0,Y 266.647,Z 392.764,A -85,B 0,C 180,E1 -18780.716,E2 -18780.716} C_VEL
LIN {X 0,Y 264.885,Z 445.774,A -85,B 0,C 180,E1 -18782.152,E2 -18782.152} C_VEL
LIN {X 0,Y 264.08,Z 455.955,A -85,B 0,C 180,E1 -18782.582,E2 -18782.582} C_VEL
LIN {X 0,Y 262.946,Z 466.081,A -85,B 0,C 180,E1 -18783.191,E2 -18783.191} C_VEL
LIN {X 0,Y 261.745,Z 475.153,A -85,B 0,C 180,E1 -18783.917,E2 -18783.917} C_VEL
LIN {X 0,Y 260.286,Z 484.282,A -85,B 0,C 180,E1 -18784.833,E2 -18784.833} C_VEL
LIN {X 0,Y 258.654,Z 493.275,A -85,B 0,C 180,E1 -18785.948,E2 -18785.948} C_VEL
LIN {X 0,Y 256.909,Z 502,A -85,B 0,C 180,E1 -18787.27,E2 -18787.27} C_VEL
LIN {X 0,Y 255.275,Z 509.391,A -85,B 0,C 180,E1 -18788.606,E2 -18788.606} C_VEL
LIN {X 0,Y 253.677,Z 516.609,A -85,B 0,C 180,E1 -18790.161,E2 -18790.161} C_VEL
LIN {X 0,Y 252.025,Z 524.189,A -85,B 0,C 180,E1 -18792.137,E2 -18792.137} C_VEL
LIN {X 0,Y 250.527,Z 530.506,A -85,B 0,C 180,E1 -18794.127,E2 -18794.127} C_VEL
LIN {X 0,Y 249.209,Z 535.765,A -85,B 0,C 180,E1 -18796.131,E2 -18796.131} C_VEL
LIN {X 0,Y 248.139,Z 540.898,A -85,B 0,C 180,E1 -18798.565,E2 -18798.565} C_VEL
LIN {X 0,Y 247.42,Z 544.889,A -85,B 0,C 180,E1 -18801.012,E2 -18801.012} C_VEL
LIN {X 0,Y 247.011,Z 547.842,A -85,B 0,C 180,E1 -18803.465,E2 -18803.465} C_VEL
LIN {X 0,Y 246.858,Z 550.295,A -85,B 0,C 180,E1 -18806.736,E2 -18806.736} C_VEL
LIN {X 0,Y 246.905,Z 550.888,A -85,B 0,C 180,E1 -18808.369,E2 -18808.369} C_VEL
LIN {X 0,Y 246.975,Z 551.045,A -85,B 0,C 180,E1 -18810,E2 -18810} C_VEL
LIN {X 0,Y 246.904,Z 550.888,A -85,B 0,C 180,E1 -18811.631,E2 -18811.631} C_VEL
LIN {X 0,Y 246.855,Z 550.295,A -85,B 0,C 180,E1 -18813.264,E2 -18813.264} C_VEL
LIN {X 0,Y 246.985,Z 547.842,A -85,B 0,C 180,E1 -18816.535,E2 -18816.535} C_VEL
LIN {X 0,Y 247.42,Z 544.889,A -85,B 0,C 180,E1 -18818.988,E2 -18818.988} C_VEL
LIN {X 0,Y 248.139,Z 540.898,A -85,B 0,C 180,E1 -18821.435,E2 -18821.435} C_VEL
LIN {X 0,Y 249.208,Z 535.765,A -85,B 0,C 180,E1 -18823.869,E2 -18823.869} C_VEL
LIN {X 0,Y 250.526,Z 530.506,A -85,B 0,C 180,E1 -18825.873,E2 -18825.873} C_VEL
LIN {X 0,Y 252.024,Z 524.189,A -85,B 0,C 180,E1 -18827.863,E2 -18827.863} C_VEL
LIN {X 0,Y 253.709,Z 516.61,A -85,B 0,C 180,E1 -18829.836,E2 -18829.836} C_VEL
LIN {X 0,Y 255.736,Z 507.473,A -85,B 0,C 180,E1 -18831.777,E2 -18831.777} C_VEL
LIN {X 0,Y 258.134,Z 495.977,A -85,B 0,C 180,E1 -18833.677,E2 -18833.677} C_VEL
LIN {X 0,Y 260.041,Z 485.915,A -85,B 0,C 180,E1 -18834.979,E2 -18834.979} C_VEL
LIN {X 0,Y 261.555,Z 476.158,A -85,B 0,C 180,E1 -18835.996,E2 -18835.996} C_VEL
LIN {X 0,Y 262.972,Z 466.082,A -85,B 0,C 180,E1 -18836.806,E2 -18836.806} C_VEL
LIN {X 0,Y 263.982,Z 456.795,A -85,B 0,C 180,E1 -18837.378,E2 -18837.378} C_VEL
LIN {X 0,Y 264.768,Z 446.983,A -85,B 0,C 180,E1 -18837.811,E2 -18837.811} C_VEL
LIN {X 0,Y 265.94,Z 414.076,A -85,B 0,C 180,E1 -18838.725,E2 -18838.725} C_VEL
LIN {X 0,Y 266.626,Z 392.081,A -85,B 0,C 180,E1 -18839.307,E2 -18839.307} C_VEL
LIN {X 0,Y 263.152,Z 371.873,A -85,B 0,C 180,E1 -18840.352,E2 -18840.352} C_VEL
LIN {X 0,Y 260.666,Z 360.23,A -85,B 0,C 180,E1 -18841.036,E2 -18841.036} C_VEL
LIN {X 0,Y 253.426,Z 343.621,A -85,B 0,C 180,E1 -18842.563,E2 -18842.563} C_VEL
LIN {X 0,Y 251.859,Z 340.025,A -85,B 0,C 180,E1 -18842.968,E2 -18842.968} C_VEL
LIN {X 0,Y 250.764,Z 334.689,A -85,B 0,C 180,E1 -18845.632,E2 -18845.632} C_VEL
LIN {X 0,Y 249.444,Z 328.86,A -85,B 0,C 180,E1 -18848.82,E2 -18848.82} C_VEL
LIN {X 0,Y 248.988,Z 326.982,A -85,B 0,C 180,E1 -18849.951,E2 -18849.951} C_VEL
LIN {X 0,Y 248.974,Z 326.961,A -85,B 0,C 180,E1 -18852.783,E2 -18852.783} C_VEL
LIN {X 0,Y 249.008,Z 326.968,A -85,B 0,C 180,E1 -18857.36,E2 -18857.36} C_VEL
LIN {X 0,Y 249.041,Z 326.963,A -85,B 0,C 180,E1 -18862.199,E2 -18862.199} C_VEL
LIN {X 0,Y 249.041,Z 326.938,A -85,B 0,C 180,E1 -18865.638,E2 -18865.638} C_VEL
LIN {X 0,Y 249.045,Z 326.965,A -85,B 0,C 180,E1 -18869.471,E2 -18869.471} C_VEL
LIN {X 0,Y 249.064,Z 326.927,A -85,B 0,C 180,E1 -18873.16,E2 -18873.16} C_VEL
LIN {X 0,Y 249.058,Z 326.958,A -85,B 0,C 180,E1 -18876.73,E2 -18876.73} C_VEL
LIN {X 0,Y 249.103,Z 326.922,A -85,B 0,C 180,E1 -18880.21,E2 -18880.21} C_VEL
LIN {X 0,Y 249.219,Z 326.92,A -85,B 0,C 180,E1 -18883.619,E2 -18883.619} C_VEL
LIN {X 0,Y 249.239,Z 326.908,A -85,B 0,C 180,E1 -18888.615,E2 -18888.615} C_VEL
LIN {X 0,Y 249.449,Z 326.875,A -85,B 0,C 180,E1 -18891.901,E2 -18891.901} C_VEL
LIN {X 0,Y 249.291,Z 326.933,A -85,B 0,C 180,E1 -18895.147,E2 -18895.147} C_VEL
LIN {X 0,Y 249.67,Z 326.855,A -85,B 0,C 180,E1 -18898.386,E2 -18898.386} C_VEL
LIN {X 0,Y 249.669,Z 326.846,A -85,B 0,C 180,E1 -18901.612,E2 -18901.612} C_VEL
LIN {X 0,Y 249.434,Z 326.904,A -85,B 0,C 180,E1 -18906.731,E2 -18906.731} C_VEL
LIN {X 0,Y 249.337,Z 326.881,A -85,B 0,C 180,E1 -18909.736,E2 -18909.736} C_VEL
LIN {X 0,Y 249.195,Z 326.945,A -85,B 0,C 180,E1 -18914.703,E2 -18914.703} C_VEL
LIN {X 0,Y 249.132,Z 326.919,A -85,B 0,C 180,E1 -18918.077,E2 -18918.077} C_VEL
LIN {X 0,Y 249.081,Z 326.943,A -85,B 0,C 180,E1 -18921.518,E2 -18921.518} C_VEL
LIN {X 0,Y 249.124,Z 326.938,A -85,B 0,C 180,E1 -18925.481,E2 -18925.481} C_VEL
LIN {X 0,Y 249.067,Z 326.94,A -85,B 0,C 180,E1 -18928.989,E2 -18928.989} C_VEL
LIN {X 0,Y 249.03,Z 326.958,A -85,B 0,C 180,E1 -18932.425,E2 -18932.425} C_VEL
LIN {X 0,Y 249.069,Z 326.95,A -85,B 0,C 180,E1 -18936.338,E2 -18936.338} C_VEL
LIN {X 0,Y 249.072,Z 326.94,A -85,B 0,C 180,E1 -18940.464,E2 -18940.464} C_VEL
LIN {X 0,Y 249.014,Z 326.948,A -85,B 0,C 180,E1 -18944.875,E2 -18944.875} C_VEL
LIN {X 0,Y 249.019,Z 326.905,A -85,B 0,C 180,E1 -18947.365,E2 -18947.365} C_VEL
LIN {X 0,Y 249.034,Z 326.963,A -85,B 0,C 180,E1 -18951.622,E2 -18951.622} C_VEL
LIN {X 0,Y 249.056,Z 326.922,A -85,B 0,C 180,E1 -18955.642,E2 -18955.642} C_VEL
LIN {X 0,Y 249.088,Z 327.191,A -85,B 0,C 180,E1 -18956.447,E2 -18956.447} C_VEL
LIN {X 0,Y 249.434,Z 328.503,A -85,B 0,C 180,E1 -18956.717,E2 -18956.717} C_VEL
LIN {X 0,Y 258.325,Z 344.365,A -85,B 0,C 180,E1 -18958.532,E2 -18958.532} C_VEL
LIN {X 0,Y 266.937,Z 360.544,A -85,B 0,C 180,E1 -18960.158,E2 -18960.158} C_VEL
LIN {X 0,Y 274.723,Z 372.024,A -85,B 0,C 180,E1 -18961.429,E2 -18961.429} C_VEL
LIN {X 0,Y 284.413,Z 383.614,A -85,B 0,C 180,E1 -18962.818,E2 -18962.818} C_VEL
LIN {X 0,Y 298.493,Z 397.804,A -85,B 0,C 180,E1 -18964.58,E2 -18964.58} C_VEL
LIN {X 0,Y 308.659,Z 406.812,A -85,B 0,C 180,E1 -18965.878,E2 -18965.878} C_VEL
LIN {X 0,Y 316.509,Z 413.509,A -85,B 0,C 180,E1 -18967.052,E2 -18967.052} C_VEL
LIN {X 0,Y 323.324,Z 418.888,A -85,B 0,C 180,E1 -18968.201,E2 -18968.201} C_VEL
LIN {X 0,Y 330.151,Z 424.447,A -85,B 0,C 180,E1 -18969.492,E2 -18969.492} C_VEL
LIN {X 0,Y 336.916,Z 429.545,A -85,B 0,C 180,E1 -18970.902,E2 -18970.902} C_VEL
LIN {X 0,Y 343.906,Z 434.7,A -85,B 0,C 180,E1 -18972.508,E2 -18972.508} C_VEL
LIN {X 0,Y 349.939,Z 439.014,A -85,B 0,C 180,E1 -18974.055,E2 -18974.055} C_VEL
LIN {X 0,Y 354.986,Z 442.628,A -85,B 0,C 180,E1 -18975.493,E2 -18975.493} C_VEL
LIN {X 0,Y 360.095,Z 445.73,A -85,B 0,C 180,E1 -18977.08,E2 -18977.08} C_VEL
LIN {X 0,Y 363.166,Z 447.626,A -85,B 0,C 180,E1 -18978.167,E2 -18978.167} C_VEL
LIN {X 0,Y 367.418,Z 450.839,A -85,B 0,C 180,E1 -18979.909,E2 -18979.909} C_VEL
LIN {X 0,Y 371.054,Z 453.173,A -85,B 0,C 180,E1 -18981.675,E2 -18981.675} C_VEL
LIN {X 0,Y 374.165,Z 454.787,A -85,B 0,C 180,E1 -18983.529,E2 -18983.529} C_VEL
LIN {X 0,Y 376.271,Z 455.746,A -85,B 0,C 180,E1 -18985.187,E2 -18985.187} C_VEL
LIN {X 0,Y 377.957,Z 456.268,A -85,B 0,C 180,E1 -18987.069,E2 -18987.069} C_VEL
LIN {X 0,Y 378.778,Z 456.768,A -85,B 0,C 180,E1 -18988.937,E2 -18988.937} C_VEL
LIN {X 0,Y 378.931,Z 456.696,A -85,B 0,C 180,E1 -18990,E2 -18990} C_VEL
LIN {X 0,Y 378.672,Z 456.667,A -85,B 0,C 180,E1 -18991.434,E2 -18991.434} C_VEL
LIN {X 0,Y 377.772,Z 456.125,A -85,B 0,C 180,E1 -18993.199,E2 -18993.199} C_VEL
LIN {X 0,Y 375.953,Z 455.604,A -85,B 0,C 180,E1 -18995.091,E2 -18995.091} C_VEL
LIN {X 0,Y 373.246,Z 454.357,A -85,B 0,C 180,E1 -18997.06,E2 -18997.06} C_VEL
LIN {X 0,Y 369.921,Z 452.477,A -85,B 0,C 180,E1 -18998.916,E2 -18998.916} C_VEL
LIN {X 0,Y 365.986,Z 449.832,A -85,B 0,C 180,E1 -19000.715,E2 -19000.715} C_VEL
LIN {X 0,Y 361.438,Z 446.437,A -85,B 0,C 180,E1 -19002.459,E2 -19002.459} C_VEL
LIN {X 0,Y 356.566,Z 443.683,A -85,B 0,C 180,E1 -19004.027,E2 -19004.027} C_VEL
LIN {X 0,Y 351.257,Z 439.998,A -85,B 0,C 180,E1 -19005.576,E2 -19005.576} C_VEL
LIN {X 0,Y 345.253,Z 435.605,A -85,B 0,C 180,E1 -19007.157,E2 -19007.157} C_VEL
LIN {X 0,Y 337.997,Z 430.437,A -85,B 0,C 180,E1 -19008.855,E2 -19008.855} C_VEL
LIN {X 0,Y 331.928,Z 425.743,A -85,B 0,C 180,E1 -19010.15,E2 -19010.15} C_VEL
LIN {X 0,Y 325.202,Z 420.515,A -85,B 0,C 180,E1 -19011.449,E2 -19011.449} C_VEL
LIN {X 0,Y 317.724,Z 414.527,A -85,B 0,C 180,E1 -19012.752,E2 -19012.752} C_VEL
LIN {X 0,Y 309.733,Z 407.702,A -85,B 0,C 180,E1 -19013.972,E2 -19013.972} C_VEL
LIN {X 0,Y 301.126,Z 400.135,A -85,B 0,C 180,E1 -19015.106,E2 -19015.106} C_VEL
LIN {X 0,Y 288.289,Z 387.737,A -85,B 0,C 180,E1 -19016.671,E2 -19016.671} C_VEL
LIN {X 0,Y 277.025,Z 375.067,A -85,B 0,C 180,E1 -19018.222,E2 -19018.222} C_VEL
LIN {X 0,Y 268.993,Z 363.756,A -85,B 0,C 180,E1 -19019.492,E2 -19019.492} C_VEL
LIN {X 0,Y 262.546,Z 352.605,A -85,B 0,C 180,E1 -19020.645,E2 -19020.645} C_VEL
LIN {X 0,Y 254.794,Z 337.803,A -85,B 0,C 180,E1 -19022.174,E2 -19022.174} C_VEL
LIN {X 0,Y 250.283,Z 330.179,A -85,B 0,C 180,E1 -19023.086,E2 -19023.086} C_VEL
LIN {X 0,Y 249.201,Z 327.715,A -85,B 0,C 180,E1 -19023.398,E2 -19023.398} C_VEL
LIN {X 0,Y 249.042,Z 326.988,A -85,B 0,C 180,E1 -19023.777,E2 -19023.777} C_VEL
LIN {X 0,Y 249.052,Z 326.964,A -85,B 0,C 180,E1 -19027.804,E2 -19027.804} C_VEL
LIN {X 0,Y 249.022,Z 326.915,A -85,B 0,C 180,E1 -19030.474,E2 -19030.474} C_VEL
LIN {X 0,Y 249.013,Z 326.942,A -85,B 0,C 180,E1 -19034.876,E2 -19034.876} C_VEL
LIN {X 0,Y 249.056,Z 326.958,A -85,B 0,C 180,E1 -19037.373,E2 -19037.373} C_VEL
LIN {X 0,Y 249.047,Z 326.963,A -85,B 0,C 180,E1 -19041.624,E2 -19041.624} C_VEL
LIN {X 0,Y 249.055,Z 326.937,A -85,B 0,C 180,E1 -19045.642,E2 -19045.642} C_VEL
LIN {X 0,Y 249.041,Z 326.962,A -85,B 0,C 180,E1 -19049.473,E2 -19049.473} C_VEL
LIN {X 0,Y 249.066,Z 326.93,A -85,B 0,C 180,E1 -19053.162,E2 -19053.162} C_VEL
LIN {X 0,Y 249.073,Z 326.961,A -85,B 0,C 180,E1 -19056.733,E2 -19056.733} C_VEL
LIN {X 0,Y 249.103,Z 326.919,A -85,B 0,C 180,E1 -19060.212,E2 -19060.212} C_VEL
LIN {X 0,Y 249.236,Z 326.929,A -85,B 0,C 180,E1 -19063.622,E2 -19063.622} C_VEL
LIN {X 0,Y 249.238,Z 326.903,A -85,B 0,C 180,E1 -19068.617,E2 -19068.617} C_VEL
LIN {X 0,Y 249.448,Z 326.884,A -85,B 0,C 180,E1 -19071.903,E2 -19071.903} C_VEL
LIN {X 0,Y 249.289,Z 326.932,A -85,B 0,C 180,E1 -19075.149,E2 -19075.149} C_VEL
LIN {X 0,Y 249.669,Z 326.846,A -85,B 0,C 180,E1 -19078.388,E2 -19078.388} C_VEL
LIN {X 0,Y 249.67,Z 326.855,A -85,B 0,C 180,E1 -19081.614,E2 -19081.614} C_VEL
LIN {X 0,Y 249.448,Z 326.9,A -85,B 0,C 180,E1 -19086.472,E2 -19086.472} C_VEL
LIN {X 0,Y 249.338,Z 326.88,A -85,B 0,C 180,E1 -19089.738,E2 -19089.738} C_VEL
LIN {X 0,Y 249.193,Z 326.94,A -85,B 0,C 180,E1 -19094.705,E2 -19094.705} C_VEL
LIN {X 0,Y 249.13,Z 326.912,A -85,B 0,C 180,E1 -19098.079,E2 -19098.079} C_VEL
LIN {X 0,Y 249.081,Z 326.95,A -85,B 0,C 180,E1 -19101.52,E2 -19101.52} C_VEL
LIN {X 0,Y 249.113,Z 326.929,A -85,B 0,C 180,E1 -19105.476,E2 -19105.476} C_VEL
LIN {X 0,Y 249.07,Z 326.947,A -85,B 0,C 180,E1 -19108.99,E2 -19108.99} C_VEL
LIN {X 0,Y 249.028,Z 326.951,A -85,B 0,C 180,E1 -19112.427,E2 -19112.427} C_VEL
LIN {X 0,Y 249.045,Z 326.958,A -85,B 0,C 180,E1 -19116.344,E2 -19116.344} C_VEL
LIN {X 0,Y 248.99,Z 326.954,A -85,B 0,C 180,E1 -19120.482,E2 -19120.482} C_VEL
LIN {X 0,Y 249,Z 326.968,A -85,B 0,C 180,E1 -19122.792,E2 -19122.792} C_VEL
LIN {X 0,Y 248.983,Z 326.957,A -85,B 0,C 180,E1 -19127.357,E2 -19127.357} C_VEL
LIN {X 0,Y 249.007,Z 327.131,A -85,B 0,C 180,E1 -19130.184,E2 -19130.184} C_VEL
LIN {X 0,Y 249.251,Z 328.127,A -85,B 0,C 180,E1 -19130.766,E2 -19130.766} C_VEL
LIN {X 0,Y 248.965,Z 329.805,A -85,B 0,C 180,E1 -19131.589,E2 -19131.589} C_VEL
LIN {X 0,Y 246.763,Z 332.959,A -85,B 0,C 180,E1 -19132.865,E2 -19132.865} C_VEL
LIN {X 0,Y 244.507,Z 336.117,A -85,B 0,C 180,E1 -19134.164,E2 -19134.164} C_VEL
LIN {X 0,Y 244.17,Z 337.824,A -85,B 0,C 180,E1 -19135.009,E2 -19135.009} C_VEL
LIN {X 0,Y 244.62,Z 339.726,A -85,B 0,C 180,E1 -19135.912,E2 -19135.912} C_VEL
LIN {X 0,Y 246.407,Z 343.735,A -85,B 0,C 180,E1 -19136.401,E2 -19136.401} C_VEL
LIN {X 0,Y 254.285,Z 361.514,A -85,B 0,C 180,E1 -19138.143,E2 -19138.143} C_VEL
LIN {X 0,Y 255.377,Z 364.747,A -85,B 0,C 180,E1 -19138.399,E2 -19138.399} C_VEL
LIN {X 0,Y 259.523,Z 387.261,A -85,B 0,C 180,E1 -19139.664,E2 -19139.664} C_VEL
LIN {X 0,Y 260.428,Z 394.258,A -85,B 0,C 180,E1 -19139.998,E2 -19139.998} C_VEL
LIN {X 0,Y 258.611,Z 446.207,A -85,B 0,C 180,E1 -19141.442,E2 -19141.442} C_VEL
LIN {X 0,Y 257.7,Z 456.804,A -85,B 0,C 180,E1 -19141.909,E2 -19141.909} C_VEL
LIN {X 0,Y 256.49,Z 467.176,A -85,B 0,C 180,E1 -19142.57,E2 -19142.57} C_VEL
LIN {X 0,Y 254.807,Z 478.987,A -85,B 0,C 180,E1 -19143.593,E2 -19143.593} C_VEL
LIN {X 0,Y 252.754,Z 490.379,A -85,B 0,C 180,E1 -19144.911,E2 -19144.911} C_VEL
LIN {X 0,Y 250.61,Z 500.671,A -85,B 0,C 180,E1 -19146.446,E2 -19146.446} C_VEL
LIN {X 0,Y 248.645,Z 509.196,A -85,B 0,C 180,E1 -19148.006,E2 -19148.006} C_VEL
LIN {X 0,Y 246.985,Z 516.415,A -85,B 0,C 180,E1 -19149.6,E2 -19149.6} C_VEL
LIN {X 0,Y 245.679,Z 522.477,A -85,B 0,C 180,E1 -19151.182,E2 -19151.182} C_VEL
LIN {X 0,Y 243.953,Z 529.155,A -85,B 0,C 180,E1 -19153.257,E2 -19153.257} C_VEL
LIN {X 0,Y 242.82,Z 533.656,A -85,B 0,C 180,E1 -19154.901,E2 -19154.901} C_VEL
LIN {X 0,Y 241.471,Z 539.148,A -85,B 0,C 180,E1 -19157.392,E2 -19157.392} C_VEL
LIN {X 0,Y 240.612,Z 543.477,A -85,B 0,C 180,E1 -19159.907,E2 -19159.907} C_VEL
LIN {X 0,Y 240.213,Z 545.846,A -85,B 0,C 180,E1 -19161.588,E2 -19161.588} C_VEL
LIN {X 0,Y 239.929,Z 547.648,A -85,B 0,C 180,E1 -19163.271,E2 -19163.271} C_VEL
LIN {X 0,Y 239.764,Z 550.101,A -85,B 0,C 180,E1 -19166.639,E2 -19166.639} C_VEL
LIN {X 0,Y 239.816,Z 550.694,A -85,B 0,C 180,E1 -19168.321,E2 -19168.321} C_VEL
LIN {X 0,Y 239.884,Z 550.851,A -85,B 0,C 180,E1 -19170,E2 -19170} C_VEL
LIN {X 0,Y 239.816,Z 550.694,A -85,B 0,C 180,E1 -19171.679,E2 -19171.679} C_VEL
LIN {X 0,Y 239.762,Z 550.101,A -85,B 0,C 180,E1 -19173.361,E2 -19173.361} C_VEL
LIN {X 0,Y 239.91,Z 547.647,A -85,B 0,C 180,E1 -19176.729,E2 -19176.729} C_VEL
LIN {X 0,Y 240.385,Z 544.694,A -85,B 0,C 180,E1 -19179.253,E2 -19179.253} C_VEL
LIN {X 0,Y 241.159,Z 540.703,A -85,B 0,C 180,E1 -19181.771,E2 -19181.771} C_VEL
LIN {X 0,Y 242.294,Z 535.571,A -85,B 0,C 180,E1 -19184.273,E2 -19184.273} C_VEL
LIN {X 0,Y 243.682,Z 530.311,A -85,B 0,C 180,E1 -19186.331,E2 -19186.331} C_VEL
LIN {X 0,Y 245.261,Z 523.995,A -85,B 0,C 180,E1 -19188.373,E2 -19188.373} C_VEL
LIN {X 0,Y 246.637,Z 518.043,A -85,B 0,C 180,E1 -19189.995,E2 -19189.995} C_VEL
LIN {X 0,Y 248.206,Z 511.115,A -85,B 0,C 180,E1 -19191.598,E2 -19191.598} C_VEL
LIN {X 0,Y 250.132,Z 502.94,A -85,B 0,C 180,E1 -19193.163,E2 -19193.163} C_VEL
LIN {X 0,Y 251.918,Z 494.432,A -85,B 0,C 180,E1 -19194.518,E2 -19194.518} C_VEL
LIN {X 0,Y 253.598,Z 485.72,A -85,B 0,C 180,E1 -19195.659,E2 -19195.659} C_VEL
LIN {X 0,Y 255.191,Z 475.964,A -85,B 0,C 180,E1 -19196.695,E2 -19196.695} C_VEL
LIN {X 0,Y 256.661,Z 465.889,A -85,B 0,C 180,E1 -19197.521,E2 -19197.521} C_VEL
LIN {X 0,Y 257.698,Z 456.8,A -85,B 0,C 180,E1 -19198.091,E2 -19198.091} C_VEL
LIN {X 0,Y 258.476,Z 447.425,A -85,B 0,C 180,E1 -19198.522,E2 -19198.522} C_VEL
LIN {X 0,Y 259.561,Z 420.818,A -85,B 0,C 180,E1 -19199.284,E2 -19199.284} C_VEL
LIN {X 0,Y 260.363,Z 392.554,A -85,B 0,C 180,E1 -19200.063,E2 -19200.063} C_VEL
LIN {X 0,Y 256.496,Z 370.306,A -85,B 0,C 180,E1 -19201.27,E2 -19201.27} C_VEL
LIN {X 0,Y 254.703,Z 362.528,A -85,B 0,C 180,E1 -19201.766,E2 -19201.766} C_VEL
LIN {X 0,Y 247.696,Z 346.632,A -85,B 0,C 180,E1 -19203.305,E2 -19203.305} C_VEL
LIN {X 0,Y 244.59,Z 339.79,A -85,B 0,C 180,E1 -19204.08,E2 -19204.08} C_VEL
LIN {X 0,Y 244.096,Z 337.524,A -85,B 0,C 180,E1 -19205.157,E2 -19205.157} C_VEL
LIN {X 0,Y 242.809,Z 331.414,A -85,B 0,C 180,E1 -19208.6,E2 -19208.6} C_VEL
LIN {X 0,Y 241.912,Z 327.834,A -85,B 0,C 180,E1 -19210.804,E2 -19210.804} C_VEL
LIN {X 0,Y 241.909,Z 327.85,A -85,B 0,C 180,E1 -19214.206,E2 -19214.206} C_VEL
LIN {X 0,Y 241.929,Z 327.849,A -85,B 0,C 180,E1 -19218.075,E2 -19218.075} C_VEL
LIN {X 0,Y 241.987,Z 327.843,A -85,B 0,C 180,E1 -19222.417,E2 -19222.417} C_VEL
LIN {X 0,Y 241.978,Z 327.818,A -85,B 0,C 180,E1 -19226.506,E2 -19226.506} C_VEL
LIN {X 0,Y 242.011,Z 327.832,A -85,B 0,C 180,E1 -19230.596,E2 -19230.596} C_VEL
LIN {X 0,Y 242.065,Z 327.802,A -85,B 0,C 180,E1 -19234.182,E2 -19234.182} C_VEL
LIN {X 0,Y 242.023,Z 327.831,A -85,B 0,C 180,E1 -19238.312,E2 -19238.312} C_VEL
LIN {X 0,Y 242.16,Z 327.794,A -85,B 0,C 180,E1 -19243.277,E2 -19243.277} C_VEL
LIN {X 0,Y 242.176,Z 327.793,A -85,B 0,C 180,E1 -19248.278,E2 -19248.278} C_VEL
LIN {X 0,Y 242.395,Z 327.75,A -85,B 0,C 180,E1 -19251.664,E2 -19251.664} C_VEL
LIN {X 0,Y 242.252,Z 327.808,A -85,B 0,C 180,E1 -19255.006,E2 -19255.006} C_VEL
LIN {X 0,Y 242.63,Z 327.731,A -85,B 0,C 180,E1 -19258.339,E2 -19258.339} C_VEL
LIN {X 0,Y 242.63,Z 327.722,A -85,B 0,C 180,E1 -19261.659,E2 -19261.659} C_VEL
LIN {X 0,Y 242.414,Z 327.78,A -85,B 0,C 180,E1 -19266.703,E2 -19266.703} C_VEL
LIN {X 0,Y 242.262,Z 327.762,A -85,B 0,C 180,E1 -19270.023,E2 -19270.023} C_VEL
LIN {X 0,Y 242.158,Z 327.82,A -85,B 0,C 180,E1 -19275.14,E2 -19275.14} C_VEL
LIN {X 0,Y 242.066,Z 327.794,A -85,B 0,C 180,E1 -19278.624,E2 -19278.624} C_VEL
LIN {X 0,Y 242.007,Z 327.834,A -85,B 0,C 180,E1 -19282.179,E2 -19282.179} C_VEL
LIN {X 0,Y 242.061,Z 327.811,A -85,B 0,C 180,E1 -19285.838,E2 -19285.838} C_VEL
LIN {X 0,Y 242.001,Z 327.828,A -85,B 0,C 180,E1 -19289.583,E2 -19289.583} C_VEL
LIN {X 0,Y 241.985,Z 327.822,A -85,B 0,C 180,E1 -19293.491,E2 -19293.491} C_VEL
LIN {X 0,Y 242.008,Z 327.841,A -85,B 0,C 180,E1 -19297.577,E2 -19297.577} C_VEL
LIN {X 0,Y 241.979,Z 327.83,A -85,B 0,C 180,E1 -19301.912,E2 -19301.912} C_VEL
LIN {X 0,Y 241.937,Z 327.806,A -85,B 0,C 180,E1 -19305.801,E2 -19305.801} C_VEL
LIN {X 0,Y 241.968,Z 327.806,A -85,B 0,C 180,E1 -19310.284,E2 -19310.284} C_VEL
LIN {X 0,Y 242.032,Z 327.799,A -85,B 0,C 180,E1 -19314.498,E2 -19314.498} C_VEL
LIN {X 0,Y 242.075,Z 328.079,A -85,B 0,C 180,E1 -19315.365,E2 -19315.365} C_VEL
LIN {X 0,Y 242.432,Z 329.422,A -85,B 0,C 180,E1 -19315.649,E2 -19315.649} C_VEL
LIN {X 0,Y 251.691,Z 345.562,A -85,B 0,C 180,E1 -19317.635,E2 -19317.635} C_VEL
LIN {X 0,Y 261.635,Z 364.556,A -85,B 0,C 180,E1 -19319.61,E2 -19319.61} C_VEL
LIN {X 0,Y 269.499,Z 376.263,A -85,B 0,C 180,E1 -19320.944,E2 -19320.944} C_VEL
LIN {X 0,Y 278.42,Z 387.227,A -85,B 0,C 180,E1 -19322.281,E2 -19322.281} C_VEL
LIN {X 0,Y 292.237,Z 401.44,A -85,B 0,C 180,E1 -19324.089,E2 -19324.089} C_VEL
LIN {X 0,Y 304.961,Z 412.701,A -85,B 0,C 180,E1 -19325.62,E2 -19325.62} C_VEL
LIN {X 0,Y 314.674,Z 420.798,A -85,B 0,C 180,E1 -19327.007,E2 -19327.007} C_VEL
LIN {X 0,Y 322.047,Z 426.596,A -85,B 0,C 180,E1 -19328.224,E2 -19328.224} C_VEL
LIN {X 0,Y 328.858,Z 431.824,A -85,B 0,C 180,E1 -19329.489,E2 -19329.489} C_VEL
LIN {X 0,Y 336.539,Z 437.613,A -85,B 0,C 180,E1 -19331.089,E2 -19331.089} C_VEL
LIN {X 0,Y 343.39,Z 442.39,A -85,B 0,C 180,E1 -19332.665,E2 -19332.665} C_VEL
LIN {X 0,Y 350.443,Z 447.518,A -85,B 0,C 180,E1 -19334.508,E2 -19334.508} C_VEL
LIN {X 0,Y 356.159,Z 451.281,A -85,B 0,C 180,E1 -19336.192,E2 -19336.192} C_VEL
LIN {X 0,Y 361.265,Z 454.246,A -85,B 0,C 180,E1 -19337.912,E2 -19337.912} C_VEL
LIN {X 0,Y 365.587,Z 457.557,A -85,B 0,C 180,E1 -19339.678,E2 -19339.678} C_VEL
LIN {X 0,Y 369.47,Z 460.039,A -85,B 0,C 180,E1 -19341.541,E2 -19341.541} C_VEL
LIN {X 0,Y 372.793,Z 461.752,A -85,B 0,C 180,E1 -19343.505,E2 -19343.505} C_VEL
LIN {X 0,Y 374.923,Z 462.692,A -85,B 0,C 180,E1 -19345.17,E2 -19345.17} C_VEL
LIN {X 0,Y 376.632,Z 463.237,A -85,B 0,C 180,E1 -19347.059,E2 -19347.059} C_VEL
LIN {X 0,Y 377.445,Z 463.741,A -85,B 0,C 180,E1 -19348.933,E2 -19348.933} C_VEL
LIN {X 0,Y 377.608,Z 463.672,A -85,B 0,C 180,E1 -19350,E2 -19350} C_VEL
LIN {X 0,Y 377.312,Z 463.608,A -85,B 0,C 180,E1 -19351.601,E2 -19351.601} C_VEL
LIN {X 0,Y 376.472,Z 463.106,A -85,B 0,C 180,E1 -19353.21,E2 -19353.21} C_VEL
LIN {X 0,Y 374.606,Z 462.564,A -85,B 0,C 180,E1 -19355.109,E2 -19355.109} C_VEL
LIN {X 0,Y 371.873,Z 461.321,A -85,B 0,C 180,E1 -19357.086,E2 -19357.086} C_VEL
LIN {X 0,Y 368.33,Z 459.337,A -85,B 0,C 180,E1 -19359.036,E2 -19359.036} C_VEL
LIN {X 0,Y 364.355,Z 456.711,A -85,B 0,C 180,E1 -19360.841,E2 -19360.841} C_VEL
LIN {X 0,Y 359.991,Z 453.359,A -85,B 0,C 180,E1 -19362.546,E2 -19362.546} C_VEL
LIN {X 0,Y 354.469,Z 450.223,A -85,B 0,C 180,E1 -19364.32,E2 -19364.32} C_VEL
LIN {X 0,Y 348.538,Z 446.126,A -85,B 0,C 180,E1 -19366.013,E2 -19366.013} C_VEL
LIN {X 0,Y 342.475,Z 441.781,A -85,B 0,C 180,E1 -19367.556,E2 -19367.556} C_VEL
LIN {X 0,Y 335.202,Z 436.647,A -85,B 0,C 180,E1 -19369.2,E2 -19369.2} C_VEL
LIN {X 0,Y 329,Z 431.917,A -85,B 0,C 180,E1 -19370.484,E2 -19370.484} C_VEL
LIN {X 0,Y 321.966,Z 426.531,A -85,B 0,C 180,E1 -19371.791,E2 -19371.791} C_VEL
LIN {X 0,Y 312.401,Z 418.934,A -85,B 0,C 180,E1 -19373.345,E2 -19373.345} C_VEL
LIN {X 0,Y 302.888,Z 410.968,A -85,B 0,C 180,E1 -19374.637,E2 -19374.637} C_VEL
LIN {X 0,Y 290.471,Z 399.681,A -85,B 0,C 180,E1 -19376.13,E2 -19376.13} C_VEL
LIN {X 0,Y 278.014,Z 386.712,A -85,B 0,C 180,E1 -19377.778,E2 -19377.778} C_VEL
LIN {X 0,Y 269.843,Z 376.732,A -85,B 0,C 180,E1 -19379.001,E2 -19379.001} C_VEL
LIN {X 0,Y 261.782,Z 364.817,A -85,B 0,C 180,E1 -19380.363,E2 -19380.363} C_VEL
LIN {X 0,Y 254.206,Z 350.409,A -85,B 0,C 180,E1 -19381.845,E2 -19381.845} C_VEL
LIN {X 0,Y 245.442,Z 334.707,A -85,B 0,C 180,E1 -19383.675,E2 -19383.675} C_VEL
LIN {X 0,Y 243.429,Z 331.292,A -85,B 0,C 180,E1 -19384.113,E2 -19384.113} C_VEL
LIN {X 0,Y 242.163,Z 328.534,A -85,B 0,C 180,E1 -19384.491,E2 -19384.491} C_VEL
LIN {X 0,Y 242.025,Z 327.847,A -85,B 0,C 180,E1 -19384.936,E2 -19384.936} C_VEL
LIN {X 0,Y 242.003,Z 327.838,A -85,B 0,C 180,E1 -19388.364,E2 -19388.364} C_VEL
LIN {X 0,Y 241.943,Z 327.784,A -85,B 0,C 180,E1 -19391.92,E2 -19391.92} C_VEL
LIN {X 0,Y 241.985,Z 327.843,A -85,B 0,C 180,E1 -19396.557,E2 -19396.557} C_VEL
LIN {X 0,Y 242.002,Z 327.825,A -85,B 0,C 180,E1 -19400.291,E2 -19400.291} C_VEL
LIN {X 0,Y 242.031,Z 327.816,A -85,B 0,C 180,E1 -19404.498,E2 -19404.498} C_VEL
LIN {X 0,Y 241.969,Z 327.845,A -85,B 0,C 180,E1 -19408.48,E2 -19408.48} C_VEL
LIN {X 0,Y 241.996,Z 327.809,A -85,B 0,C 180,E1 -19412.312,E2 -19412.312} C_VEL
LIN {X 0,Y 242.051,Z 327.833,A -85,B 0,C 180,E1 -19416.016,E2 -19416.016} C_VEL
LIN {X 0,Y 242.03,Z 327.804,A -85,B 0,C 180,E1 -19419.608,E2 -19419.608} C_VEL
LIN {X 0,Y 242.158,Z 327.805,A -85,B 0,C 180,E1 -19423.279,E2 -19423.279} C_VEL
LIN {X 0,Y 242.174,Z 327.786,A -85,B 0,C 180,E1 -19428.28,E2 -19428.28} C_VEL
LIN {X 0,Y 242.394,Z 327.758,A -85,B 0,C 180,E1 -19431.665,E2 -19431.665} C_VEL
LIN {X 0,Y 242.25,Z 327.809,A -85,B 0,C 180,E1 -19435.008,E2 -19435.008} C_VEL
LIN {X 0,Y 242.63,Z 327.722,A -85,B 0,C 180,E1 -19438.341,E2 -19438.341} C_VEL
LIN {X 0,Y 242.63,Z 327.731,A -85,B 0,C 180,E1 -19441.661,E2 -19441.661} C_VEL
LIN {X 0,Y 242.418,Z 327.774,A -85,B 0,C 180,E1 -19446.66,E2 -19446.66} C_VEL
LIN {X 0,Y 242.263,Z 327.761,A -85,B 0,C 180,E1 -19450.025,E2 -19450.025} C_VEL
LIN {X 0,Y 242.152,Z 327.814,A -85,B 0,C 180,E1 -19455.143,E2 -19455.143} C_VEL
LIN {X 0,Y 242.065,Z 327.79,A -85,B 0,C 180,E1 -19458.626,E2 -19458.626} C_VEL
LIN {X 0,Y 242.003,Z 327.835,A -85,B 0,C 180,E1 -19462.182,E2 -19462.182} C_VEL
LIN {X 0,Y 242.064,Z 327.802,A -85,B 0,C 180,E1 -19465.839,E2 -19465.839} C_VEL
LIN {X 0,Y 242.005,Z 327.836,A -85,B 0,C 180,E1 -19469.585,E2 -19469.585} C_VEL
LIN {X 0,Y 241.978,Z 327.818,A -85,B 0,C 180,E1 -19473.494,E2 -19473.494} C_VEL
LIN {X 0,Y 241.987,Z 327.843,A -85,B 0,C 180,E1 -19477.583,E2 -19477.583} C_VEL
LIN {X 0,Y 241.929,Z 327.848,A -85,B 0,C 180,E1 -19481.925,E2 -19481.925} C_VEL
LIN {X 0,Y 241.908,Z 327.853,A -85,B 0,C 180,E1 -19486.579,E2 -19486.579} C_VEL
LIN {X 0,Y 241.943,Z 327.944,A -85,B 0,C 180,E1 -19489.332,E2 -19489.332} C_VEL
LIN {X 0,Y 243.615,Z 334.896,A -85,B 0,C 180,E1 -19493.385,E2 -19493.385} C_VEL
LIN {X 0,Y 244.17,Z 337.824,A -85,B 0,C 180,E1 -19495.009,E2 -19495.009} C_VEL
LIN {X 0,Y 244.808,Z 339.945,A -85,B 0,C 180,E1 -19495.718,E2 -19495.718} C_VEL
LIN {X 0,Y 245.829,Z 342.897,A -85,B 0,C 180,E1 -19496.228,E2 -19496.228} C_VEL
LIN {X 0,Y 247.473,Z 348.21,A -85,B 0,C 180,E1 -19496.715,E2 -19496.715} C_VEL
LIN {X 0,Y 248.439,Z 354.256,A -85,B 0,C 180,E1 -19497.049,E2 -19497.049} C_VEL
LIN {X 0,Y 249.49,Z 366.89,A -85,B 0,C 180,E1 -19497.641,E2 -19497.641} C_VEL
LIN {X 0,Y 253.391,Z 388.37,A -85,B 0,C 180,E1 -19498.892,E2 -19498.892} C_VEL
LIN {X 0,Y 254.253,Z 395.105,A -85,B 0,C 180,E1 -19499.225,E2 -19499.225} C_VEL
LIN {X 0,Y 252.404,Z 445.476,A -85,B 0,C 180,E1 -19500.648,E2 -19500.648} C_VEL
LIN {X 0,Y 251.536,Z 455.997,A -85,B 0,C 180,E1 -19501.117,E2 -19501.117} C_VEL
LIN {X 0,Y 250.384,Z 465.695,A -85,B 0,C 180,E1 -19501.728,E2 -19501.728} C_VEL
LIN {X 0,Y 248.914,Z 475.772,A -85,B 0,C 180,E1 -19502.576,E2 -19502.576} C_VEL
LIN {X 0,Y 247.219,Z 485.526,A -85,B 0,C 180,E1 -19503.629,E2 -19503.629} C_VEL
LIN {X 0,Y 245.183,Z 495.589,A -85,B 0,C 180,E1 -19504.989,E2 -19504.989} C_VEL
LIN {X 0,Y 242.565,Z 507.084,A -85,B 0,C 180,E1 -19506.975,E2 -19506.975} C_VEL
LIN {X 0,Y 240.304,Z 516.22,A -85,B 0,C 180,E1 -19509.007,E2 -19509.007} C_VEL
LIN {X 0,Y 238.846,Z 522.594,A -85,B 0,C 180,E1 -19510.724,E2 -19510.724} C_VEL
LIN {X 0,Y 237.112,Z 528.96,A -85,B 0,C 180,E1 -19512.759,E2 -19512.759} C_VEL
LIN {X 0,Y 235.942,Z 533.461,A -85,B 0,C 180,E1 -19514.45,E2 -19514.45} C_VEL
LIN {X 0,Y 234.515,Z 538.953,A -85,B 0,C 180,E1 -19517.011,E2 -19517.011} C_VEL
LIN {X 0,Y 233.584,Z 543.281,A -85,B 0,C 180,E1 -19519.6,E2 -19519.6} C_VEL
LIN {X 0,Y 233.18,Z 545.652,A -85,B 0,C 180,E1 -19521.333,E2 -19521.333} C_VEL
LIN {X 0,Y 232.874,Z 547.454,A -85,B 0,C 180,E1 -19523.067,E2 -19523.067} C_VEL
LIN {X 0,Y 232.674,Z 549.907,A -85,B 0,C 180,E1 -19526.537,E2 -19526.537} C_VEL
LIN {X 0,Y 232.729,Z 550.5,A -85,B 0,C 180,E1 -19528.27,E2 -19528.27} C_VEL
LIN {X 0,Y 232.795,Z 550.657,A -85,B 0,C 180,E1 -19530,E2 -19530} C_VEL
LIN {X 0,Y 232.729,Z 550.5,A -85,B 0,C 180,E1 -19531.73,E2 -19531.73} C_VEL
LIN {X 0,Y 232.689,Z 549.229,A -85,B 0,C 180,E1 -19534.637,E2 -19534.637} C_VEL
LIN {X 0,Y 232.833,Z 547.453,A -85,B 0,C 180,E1 -19536.935,E2 -19536.935} C_VEL
LIN {X 0,Y 233.369,Z 544.5,A -85,B 0,C 180,E1 -19539.534,E2 -19539.534} C_VEL
LIN {X 0,Y 234.173,Z 540.508,A -85,B 0,C 180,E1 -19542.127,E2 -19542.127} C_VEL
LIN {X 0,Y 235.397,Z 535.376,A -85,B 0,C 180,E1 -19544.701,E2 -19544.701} C_VEL
LIN {X 0,Y 236.852,Z 530.117,A -85,B 0,C 180,E1 -19546.816,E2 -19546.816} C_VEL
LIN {X 0,Y 238.518,Z 523.801,A -85,B 0,C 180,E1 -19548.912,E2 -19548.912} C_VEL
LIN {X 0,Y 239.94,Z 517.848,A -85,B 0,C 180,E1 -19550.578,E2 -19550.578} C_VEL
LIN {X 0,Y 241.61,Z 510.921,A -85,B 0,C 180,E1 -19552.218,E2 -19552.218} C_VEL
LIN {X 0,Y 243.585,Z 502.745,A -85,B 0,C 180,E1 -19553.824,E2 -19553.824} C_VEL
LIN {X 0,Y 245.481,Z 494.238,A -85,B 0,C 180,E1 -19555.205,E2 -19555.205} C_VEL
LIN {X 0,Y 247.221,Z 485.526,A -85,B 0,C 180,E1 -19556.371,E2 -19556.371} C_VEL
LIN {X 0,Y 248.884,Z 475.771,A -85,B 0,C 180,E1 -19557.427,E2 -19557.427} C_VEL
LIN {X 0,Y 250.375,Z 465.694,A -85,B 0,C 180,E1 -19558.273,E2 -19558.273} C_VEL
LIN {X 0,Y 251.54,Z 455.993,A -85,B 0,C 180,E1 -19558.883,E2 -19558.883} C_VEL
LIN {X 0,Y 252.31,Z 446.622,A -85,B 0,C 180,E1 -19559.312,E2 -19559.312} C_VEL
LIN {X 0,Y 253.537,Z 414.773,A -85,B 0,C 180,E1 -19560.238,E2 -19560.238} C_VEL
LIN {X 0,Y 254.273,Z 393.938,A -85,B 0,C 180,E1 -19560.81,E2 -19560.81} C_VEL
LIN {X 0,Y 250.515,Z 372.092,A -85,B 0,C 180,E1 -19562.04,E2 -19562.04} C_VEL
LIN {X 0,Y 249.144,Z 365.785,A -85,B 0,C 180,E1 -19562.446,E2 -19562.446} C_VEL
LIN {X 0,Y 241.301,Z 347.845,A -85,B 0,C 180,E1 -19564.258,E2 -19564.258} C_VEL
LIN {X 0,Y 237.363,Z 339.681,A -85,B 0,C 180,E1 -19565.249,E2 -19565.249} C_VEL
LIN {X 0,Y 236.869,Z 337.291,A -85,B 0,C 180,E1 -19566.398,E2 -19566.398} C_VEL
LIN {X 0,Y 235.342,Z 330.8,A -85,B 0,C 180,E1 -19570.272,E2 -19570.272} C_VEL
LIN {X 0,Y 234.862,Z 328.711,A -85,B 0,C 180,E1 -19571.683,E2 -19571.683} C_VEL
LIN {X 0,Y 234.882,Z 328.716,A -85,B 0,C 180,E1 -19575.898,E2 -19575.898} C_VEL
LIN {X 0,Y 234.871,Z 328.718,A -85,B 0,C 180,E1 -19578.828,E2 -19578.828} C_VEL
LIN {X 0,Y 234.926,Z 328.721,A -85,B 0,C 180,E1 -19583.249,E2 -19583.249} C_VEL
LIN {X 0,Y 234.954,Z 328.7,A -85,B 0,C 180,E1 -19587.423,E2 -19587.423} C_VEL
LIN {X 0,Y 234.933,Z 328.701,A -85,B 0,C 180,E1 -19591.402,E2 -19591.402} C_VEL
LIN {X 0,Y 234.975,Z 328.699,A -85,B 0,C 180,E1 -19595.244,E2 -19595.244} C_VEL
LIN {X 0,Y 234.994,Z 328.695,A -85,B 0,C 180,E1 -19598.967,E2 -19598.967} C_VEL
LIN {X 0,Y 235.092,Z 328.67,A -85,B 0,C 180,E1 -19603.059,E2 -19603.059} C_VEL
LIN {X 0,Y 235.109,Z 328.679,A -85,B 0,C 180,E1 -19607.921,E2 -19607.921} C_VEL
LIN {X 0,Y 235.326,Z 328.627,A -85,B 0,C 180,E1 -19611.411,E2 -19611.411} C_VEL
LIN {X 0,Y 235.368,Z 328.649,A -85,B 0,C 180,E1 -19613.139,E2 -19613.139} C_VEL
LIN {X 0,Y 235.59,Z 328.608,A -85,B 0,C 180,E1 -19618.29,E2 -19618.29} C_VEL
LIN {X 0,Y 235.589,Z 328.599,A -85,B 0,C 180,E1 -19621.709,E2 -19621.709} C_VEL
LIN {X 0,Y 235.367,Z 328.656,A -85,B 0,C 180,E1 -19626.859,E2 -19626.859} C_VEL
LIN {X 0,Y 235.209,Z 328.64,A -85,B 0,C 180,E1 -19630.327,E2 -19630.327} C_VEL
LIN {X 0,Y 235.106,Z 328.696,A -85,B 0,C 180,E1 -19635.606,E2 -19635.606} C_VEL
LIN {X 0,Y 235.002,Z 328.672,A -85,B 0,C 180,E1 -19639.205,E2 -19639.205} C_VEL
LIN {X 0,Y 234.955,Z 328.717,A -85,B 0,C 180,E1 -19642.882,E2 -19642.882} C_VEL
LIN {X 0,Y 234.962,Z 328.686,A -85,B 0,C 180,E1 -19646.657,E2 -19646.657} C_VEL
LIN {X 0,Y 234.917,Z 328.722,A -85,B 0,C 180,E1 -19650.569,E2 -19650.569} C_VEL
LIN {X 0,Y 234.955,Z 328.692,A -85,B 0,C 180,E1 -19654.633,E2 -19654.633} C_VEL
LIN {X 0,Y 234.961,Z 328.71,A -85,B 0,C 180,E1 -19658.952,E2 -19658.952} C_VEL
LIN {X 0,Y 234.959,Z 328.718,A -85,B 0,C 180,E1 -19663.468,E2 -19663.468} C_VEL
LIN {X 0,Y 234.891,Z 328.662,A -85,B 0,C 180,E1 -19668.416,E2 -19668.416} C_VEL
LIN {X 0,Y 234.95,Z 328.697,A -85,B 0,C 180,E1 -19671.086,E2 -19671.086} C_VEL
LIN {X 0,Y 235.005,Z 328.93,A -85,B 0,C 180,E1 -19674.157,E2 -19674.157} C_VEL
LIN {X 0,Y 235.259,Z 329.92,A -85,B 0,C 180,E1 -19674.445,E2 -19674.445} C_VEL
LIN {X 0,Y 236.921,Z 332.766,A -85,B 0,C 180,E1 -19674.86,E2 -19674.86} C_VEL
LIN {X 0,Y 247.643,Z 351.762,A -85,B 0,C 180,E1 -19677.245,E2 -19677.245} C_VEL
LIN {X 0,Y 256.195,Z 368.268,A -85,B 0,C 180,E1 -19679.008,E2 -19679.008} C_VEL
LIN {X 0,Y 263.798,Z 379.807,A -85,B 0,C 180,E1 -19680.358,E2 -19680.358} C_VEL
LIN {X 0,Y 270.747,Z 388.716,A -85,B 0,C 180,E1 -19681.462,E2 -19681.462} C_VEL
LIN {X 0,Y 283.005,Z 402.085,A -85,B 0,C 180,E1 -19683.187,E2 -19683.187} C_VEL
LIN {X 0,Y 294.128,Z 412.447,A -85,B 0,C 180,E1 -19684.561,E2 -19684.561} C_VEL
LIN {X 0,Y 303.448,Z 420.406,A -85,B 0,C 180,E1 -19685.672,E2 -19685.672} C_VEL
LIN {X 0,Y 313.037,Z 428.22,A -85,B 0,C 180,E1 -19686.996,E2 -19686.996} C_VEL
LIN {X 0,Y 320.757,Z 434.248,A -85,B 0,C 180,E1 -19688.268,E2 -19688.268} C_VEL
LIN {X 0,Y 328.405,Z 439.801,A -85,B 0,C 180,E1 -19689.702,E2 -19689.702} C_VEL
LIN {X 0,Y 336.246,Z 445.804,A -85,B 0,C 180,E1 -19691.374,E2 -19691.374} C_VEL
LIN {X 0,Y 343.934,Z 451.025,A -85,B 0,C 180,E1 -19693.203,E2 -19693.203} C_VEL
LIN {X 0,Y 350.182,Z 455.573,A -85,B 0,C 180,E1 -19694.921,E2 -19694.921} C_VEL
LIN {X 0,Y 356.013,Z 459.149,A -85,B 0,C 180,E1 -19696.71,E2 -19696.71} C_VEL
LIN {X 0,Y 358.954,Z 460.86,A -85,B 0,C 180,E1 -19697.717,E2 -19697.717} C_VEL
LIN {X 0,Y 363.331,Z 464.187,A -85,B 0,C 180,E1 -19699.493,E2 -19699.493} C_VEL
LIN {X 0,Y 366.919,Z 466.51,A -85,B 0,C 180,E1 -19701.186,E2 -19701.186} C_VEL
LIN {X 0,Y 369.069,Z 467.663,A -85,B 0,C 180,E1 -19702.34,E2 -19702.34} C_VEL
LIN {X 0,Y 370.864,Z 468.58,A -85,B 0,C 180,E1 -19703.471,E2 -19703.471} C_VEL
LIN {X 0,Y 372.392,Z 469.215,A -85,B 0,C 180,E1 -19704.585,E2 -19704.585} C_VEL
LIN {X 0,Y 373.636,Z 469.686,A -85,B 0,C 180,E1 -19705.685,E2 -19705.685} C_VEL
LIN {X 0,Y 374.611,Z 469.972,A -85,B 0,C 180,E1 -19706.774,E2 -19706.774} C_VEL
LIN {X 0,Y 375.249,Z 470.329,A -85,B 0,C 180,E1 -19707.853,E2 -19707.853} C_VEL
LIN {X 0,Y 375.619,Z 470.574,A -85,B 0,C 180,E1 -19708.928,E2 -19708.928} C_VEL
LIN {X 0,Y 375.784,Z 470.522,A -85,B 0,C 180,E1 -19710,E2 -19710} C_VEL
LIN {X 0,Y 375.639,Z 470.517,A -85,B 0,C 180,E1 -19711.072,E2 -19711.072} C_VEL
LIN {X 0,Y 375.268,Z 470.287,A -85,B 0,C 180,E1 -19712.147,E2 -19712.147} C_VEL
LIN {X 0,Y 374.624,Z 469.961,A -85,B 0,C 180,E1 -19713.226,E2 -19713.226} C_VEL
LIN {X 0,Y 373.581,Z 469.632,A -85,B 0,C 180,E1 -19714.402,E2 -19714.402} C_VEL
LIN {X 0,Y 372.415,Z 469.225,A -85,B 0,C 180,E1 -19715.414,E2 -19715.414} C_VEL
LIN {X 0,Y 370.888,Z 468.573,A -85,B 0,C 180,E1 -19716.528,E2 -19716.528} C_VEL
LIN {X 0,Y 368.836,Z 467.568,A -85,B 0,C 180,E1 -19717.769,E2 -19717.769} C_VEL
LIN {X 0,Y 365.356,Z 465.565,A -85,B 0,C 180,E1 -19719.584,E2 -19719.584} C_VEL
LIN {X 0,Y 361.253,Z 462.689,A -85,B 0,C 180,E1 -19721.37,E2 -19721.37} C_VEL
LIN {X 0,Y 357.518,Z 459.908,A -85,B 0,C 180,E1 -19722.793,E2 -19722.793} C_VEL
LIN {X 0,Y 351.874,Z 456.649,A -85,B 0,C 180,E1 -19724.579,E2 -19724.579} C_VEL
LIN {X 0,Y 345.591,Z 452.326,A -85,B 0,C 180,E1 -19726.347,E2 -19726.347} C_VEL
LIN {X 0,Y 339.869,Z 448.222,A -85,B 0,C 180,E1 -19727.789,E2 -19727.789} C_VEL
LIN {X 0,Y 332.503,Z 443.029,A -85,B 0,C 180,E1 -19729.446,E2 -19729.446} C_VEL
LIN {X 0,Y 325.895,Z 438.075,A -85,B 0,C 180,E1 -19730.783,E2 -19730.783} C_VEL
LIN {X 0,Y 318.178,Z 432.164,A -85,B 0,C 180,E1 -19732.183,E2 -19732.183} C_VEL
LIN {X 0,Y 310.346,Z 426.141,A -85,B 0,C 180,E1 -19733.387,E2 -19733.387} C_VEL
LIN {X 0,Y 302.137,Z 419.362,A -85,B 0,C 180,E1 -19734.485,E2 -19734.485} C_VEL
LIN {X 0,Y 289.724,Z 408.61,A -85,B 0,C 180,E1 -19735.961,E2 -19735.961} C_VEL
LIN {X 0,Y 275.47,Z 394.165,A -85,B 0,C 180,E1 -19737.843,E2 -19737.843} C_VEL
LIN {X 0,Y 265.578,Z 382.314,A -85,B 0,C 180,E1 -19739.346,E2 -19739.346} C_VEL
LIN {X 0,Y 257.215,Z 369.988,A -85,B 0,C 180,E1 -19740.8,E2 -19740.8} C_VEL
LIN {X 0,Y 250.206,Z 356.901,A -85,B 0,C 180,E1 -19742.204,E2 -19742.204} C_VEL
LIN {X 0,Y 242.649,Z 342.663,A -85,B 0,C 180,E1 -19743.84,E2 -19743.84} C_VEL
LIN {X 0,Y 236.57,Z 332.343,A -85,B 0,C 180,E1 -19745.216,E2 -19745.216} C_VEL
LIN {X 0,Y 235.129,Z 329.441,A -85,B 0,C 180,E1 -19745.647,E2 -19745.647} C_VEL
LIN {X 0,Y 234.951,Z 328.731,A -85,B 0,C 180,E1 -19746.136,E2 -19746.136} C_VEL
LIN {X 0,Y 234.937,Z 328.698,A -85,B 0,C 180,E1 -19748.944,E2 -19748.944} C_VEL
LIN {X 0,Y 234.891,Z 328.67,A -85,B 0,C 180,E1 -19753.484,E2 -19753.484} C_VEL
LIN {X 0,Y 234.959,Z 328.718,A -85,B 0,C 180,E1 -19756.532,E2 -19756.532} C_VEL
LIN {X 0,Y 234.949,Z 328.713,A -85,B 0,C 180,E1 -19761.086,E2 -19761.086} C_VEL
LIN {X 0,Y 234.955,Z 328.692,A -85,B 0,C 180,E1 -19765.367,E2 -19765.367} C_VEL
LIN {X 0,Y 234.917,Z 328.722,A -85,B 0,C 180,E1 -19769.431,E2 -19769.431} C_VEL
LIN {X 0,Y 234.988,Z 328.687,A -85,B 0,C 180,E1 -19773.794,E2 -19773.794} C_VEL
LIN {X 0,Y 235.005,Z 328.687,A -85,B 0,C 180,E1 -19778.97,E2 -19778.97} C_VEL
LIN {X 0,Y 235.091,Z 328.683,A -85,B 0,C 180,E1 -19783.06,E2 -19783.06} C_VEL
LIN {X 0,Y 235.108,Z 328.671,A -85,B 0,C 180,E1 -19787.923,E2 -19787.923} C_VEL
LIN {X 0,Y 235.325,Z 328.634,A -85,B 0,C 180,E1 -19791.413,E2 -19791.413} C_VEL
LIN {X 0,Y 235.367,Z 328.656,A -85,B 0,C 180,E1 -19793.141,E2 -19793.141} C_VEL
LIN {X 0,Y 235.589,Z 328.599,A -85,B 0,C 180,E1 -19798.291,E2 -19798.291} C_VEL
LIN {X 0,Y 235.59,Z 328.608,A -85,B 0,C 180,E1 -19801.71,E2 -19801.71} C_VEL
LIN {X 0,Y 235.368,Z 328.649,A -85,B 0,C 180,E1 -19806.861,E2 -19806.861} C_VEL
LIN {X 0,Y 235.21,Z 328.641,A -85,B 0,C 180,E1 -19810.329,E2 -19810.329} C_VEL
LIN {X 0,Y 235.103,Z 328.688,A -85,B 0,C 180,E1 -19815.608,E2 -19815.608} C_VEL
LIN {X 0,Y 235.001,Z 328.671,A -85,B 0,C 180,E1 -19819.207,E2 -19819.207} C_VEL
LIN {X 0,Y 234.949,Z 328.717,A -85,B 0,C 180,E1 -19822.885,E2 -19822.885} C_VEL
LIN {X 0,Y 234.964,Z 328.682,A -85,B 0,C 180,E1 -19826.659,E2 -19826.659} C_VEL
LIN {X 0,Y 234.92,Z 328.724,A -85,B 0,C 180,E1 -19830.57,E2 -19830.57} C_VEL
LIN {X 0,Y 234.928,Z 328.696,A -85,B 0,C 180,E1 -19834.639,E2 -19834.639} C_VEL
LIN {X 0,Y 234.912,Z 328.71,A -85,B 0,C 180,E1 -19838.937,E2 -19838.937} C_VEL
LIN {X 0,Y 234.877,Z 328.72,A -85,B 0,C 180,E1 -19843.49,E2 -19843.49} C_VEL
LIN {X 0,Y 234.863,Z 328.702,A -85,B 0,C 180,E1 -19848.063,E2 -19848.063} C_VEL
LIN {X 0,Y 234.899,Z 328.946,A -85,B 0,C 180,E1 -19848.578,E2 -19848.578} C_VEL
LIN {X 0,Y 236.781,Z 336.704,A -85,B 0,C 180,E1 -19853.265,E2 -19853.265} C_VEL
LIN {X 0,Y 237.316,Z 339.45,A -85,B 0,C 180,E1 -19854.702,E2 -19854.702} C_VEL
LIN {X 0,Y 239.069,Z 343.318,A -85,B 0,C 180,E1 -19855.218,E2 -19855.218} C_VEL
LIN {X 0,Y 245.948,Z 358.114,A -85,B 0,C 180,E1 -19856.822,E2 -19856.822} C_VEL
LIN {X 0,Y 249.49,Z 366.89,A -85,B 0,C 180,E1 -19857.641,E2 -19857.641} C_VEL
LIN {X 0,Y 249.937,Z 374.648,A -85,B 0,C 180,E1 -19857.963,E2 -19857.963} C_VEL
LIN {X 0,Y 249.486,Z 382.514,A -85,B 0,C 180,E1 -19858.16,E2 -19858.16} C_VEL
LIN {X 0,Y 248.042,Z 398.357,A -85,B 0,C 180,E1 -19858.481,E2 -19858.481} C_VEL
LIN {X 0,Y 246.213,Z 445.916,A -85,B 0,C 180,E1 -19859.864,E2 -19859.864} C_VEL
LIN {X 0,Y 245.243,Z 456.796,A -85,B 0,C 180,E1 -19860.37,E2 -19860.37} C_VEL
LIN {X 0,Y 243.818,Z 468.076,A -85,B 0,C 180,E1 -19861.131,E2 -19861.131} C_VEL
LIN {X 0,Y 241.783,Z 480.435,A -85,B 0,C 180,E1 -19862.285,E2 -19862.285} C_VEL
LIN {X 0,Y 239.643,Z 491.342,A -85,B 0,C 180,E1 -19863.669,E2 -19863.669} C_VEL
LIN {X 0,Y 237.622,Z 500.282,A -85,B 0,C 180,E1 -19865.074,E2 -19865.074} C_VEL
LIN {X 0,Y 235.511,Z 508.807,A -85,B 0,C 180,E1 -19866.71,E2 -19866.71} C_VEL
LIN {X 0,Y 233.655,Z 516.025,A -85,B 0,C 180,E1 -19868.38,E2 -19868.38} C_VEL
LIN {X 0,Y 232.241,Z 521.772,A -85,B 0,C 180,E1 -19869.943,E2 -19869.943} C_VEL
LIN {X 0,Y 230.291,Z 528.764,A -85,B 0,C 180,E1 -19872.232,E2 -19872.232} C_VEL
LIN {X 0,Y 229.088,Z 533.267,A -85,B 0,C 180,E1 -19873.973,E2 -19873.973} C_VEL
LIN {X 0,Y 227.552,Z 538.758,A -85,B 0,C 180,E1 -19876.607,E2 -19876.607} C_VEL
LIN {X 0,Y 226.58,Z 543.087,A -85,B 0,C 180,E1 -19879.275,E2 -19879.275} C_VEL
LIN {X 0,Y 226.138,Z 545.458,A -85,B 0,C 180,E1 -19881.061,E2 -19881.061} C_VEL
LIN {X 0,Y 225.811,Z 547.259,A -85,B 0,C 180,E1 -19882.849,E2 -19882.849} C_VEL
LIN {X 0,Y 225.588,Z 549.713,A -85,B 0,C 180,E1 -19886.428,E2 -19886.428} C_VEL
LIN {X 0,Y 225.625,Z 550.306,A -85,B 0,C 180,E1 -19888.215,E2 -19888.215} C_VEL
LIN {X 0,Y 225.708,Z 550.464,A -85,B 0,C 180,E1 -19890,E2 -19890} C_VEL
LIN {X 0,Y 225.625,Z 550.306,A -85,B 0,C 180,E1 -19891.785,E2 -19891.785} C_VEL
LIN {X 0,Y 225.587,Z 549.239,A -85,B 0,C 180,E1 -19894.475,E2 -19894.475} C_VEL
LIN {X 0,Y 225.782,Z 547.259,A -85,B 0,C 180,E1 -19897.152,E2 -19897.152} C_VEL
LIN {X 0,Y 226.334,Z 544.305,A -85,B 0,C 180,E1 -19899.833,E2 -19899.833} C_VEL
LIN {X 0,Y 227.206,Z 540.313,A -85,B 0,C 180,E1 -19902.505,E2 -19902.505} C_VEL
LIN {X 0,Y 228.517,Z 535.182,A -85,B 0,C 180,E1 -19905.154,E2 -19905.154} C_VEL
LIN {X 0,Y 230.014,Z 529.921,A -85,B 0,C 180,E1 -19907.332,E2 -19907.332} C_VEL
LIN {X 0,Y 231.772,Z 523.606,A -85,B 0,C 180,E1 -19909.484,E2 -19909.484} C_VEL
LIN {X 0,Y 233.277,Z 517.653,A -85,B 0,C 180,E1 -19911.193,E2 -19911.193} C_VEL
LIN {X 0,Y 235.034,Z 510.726,A -85,B 0,C 180,E1 -19912.875,E2 -19912.875} C_VEL
LIN {X 0,Y 237.113,Z 502.551,A -85,B 0,C 180,E1 -19914.516,E2 -19914.516} C_VEL
LIN {X 0,Y 239.066,Z 494.044,A -85,B 0,C 180,E1 -19915.931,E2 -19915.931} C_VEL
LIN {X 0,Y 240.882,Z 485.332,A -85,B 0,C 180,E1 -19917.121,E2 -19917.121} C_VEL
LIN {X 0,Y 242.419,Z 476.583,A -85,B 0,C 180,E1 -19918.105,E2 -19918.105} C_VEL
LIN {X 0,Y 243.976,Z 466.788,A -85,B 0,C 180,E1 -19918.966,E2 -19918.966} C_VEL
LIN {X 0,Y 245.221,Z 456.804,A -85,B 0,C 180,E1 -19919.632,E2 -19919.632} C_VEL
LIN {X 0,Y 246.121,Z 447.107,A -85,B 0,C 180,E1 -19920.094,E2 -19920.094} C_VEL
LIN {X 0,Y 247.168,Z 422.872,A -85,B 0,C 180,E1 -19920.828,E2 -19920.828} C_VEL
LIN {X 0,Y 248.139,Z 394.644,A -85,B 0,C 180,E1 -19921.629,E2 -19921.629} C_VEL
LIN {X 0,Y 243.965,Z 370.441,A -85,B 0,C 180,E1 -19923.057,E2 -19923.057} C_VEL
LIN {X 0,Y 241.959,Z 364.958,A -85,B 0,C 180,E1 -19923.555,E2 -19923.555} C_VEL
LIN {X 0,Y 235.349,Z 350.278,A -85,B 0,C 180,E1 -19925.155,E2 -19925.155} C_VEL
LIN {X 0,Y 230.165,Z 339.585,A -85,B 0,C 180,E1 -19926.504,E2 -19926.504} C_VEL
LIN {X 0,Y 229.902,Z 338.338,A -85,B 0,C 180,E1 -19926.984,E2 -19926.984} C_VEL
LIN {X 0,Y 228.284,Z 331.829,A -85,B 0,C 180,E1 -19931.038,E2 -19931.038} C_VEL
